C07299=1225.069,224.559,-58.740,-177.166,6.220,148.282
C07300=1225.074,224.310,-58.716,-177.168,6.218,148.282
C07301=1225.078,224.061,-58.690,-177.171,6.216,148.282
C07302=1225.084,223.813,-58.665,-177.173,6.215,148.283
C07303=1225.088,223.563,-58.640,-177.175,6.213,148.283
C07304=1225.092,223.315,-58.615,-177.178,6.211,148.283
C07305=1225.097,223.066,-58.590,-177.181,6.209,148.284
C07306=1225.102,222.818,-58.565,-177.183,6.207,148.284
C07307=1225.105,222.569,-58.541,-177.186,6.206,148.284
C07308=1225.110,222.321,-58.515,-177.188,6.204,148.285
C07309=1225.115,222.072,-58.490,-177.191,6.202,148.285
C07310=1225.120,221.823,-58.465,-177.194,6.200,148.285
C07311=1225.124,221.575,-58.441,-177.196,6.198,148.286
C07312=1225.128,221.325,-58.416,-177.199,6.196,148.286
C07313=1225.133,221.077,-58.390,-177.201,6.195,148.286
C07314=1225.137,220.828,-58.366,-177.204,6.193,148.287
C07315=1225.142,220.579,-58.341,-177.206,6.192,148.287
C07316=1225.146,220.331,-58.315,-177.209,6.190,148.287
C07317=1225.151,220.082,-58.291,-177.212,6.188,148.288
C07318=1225.156,219.833,-58.267,-177.214,6.186,148.288
C07319=1225.160,219.584,-58.242,-177.217,6.184,148.288
C07320=1225.165,219.336,-58.217,-177.219,6.182,148.289
C07321=1225.169,219.087,-58.192,-177.222,6.180,148.289
C07322=1225.174,218.838,-58.167,-177.225,6.178,148.289
C07323=1225.178,218.590,-58.142,-177.227,6.177,148.290
C07324=1225.183,218.341,-58.117,-177.229,6.176,148.290
C07325=1225.187,218.092,-58.093,-177.232,6.174,148.290
C07326=1225.192,217.843,-58.068,-177.235,6.172,148.291
C07327=1225.197,217.594,-58.044,-177.237,6.170,148.291
C07328=1225.201,217.347,-58.019,-177.240,6.168,148.291
C07329=1225.206,217.097,-57.994,-177.243,6.166,148.292
C07330=1225.210,216.849,-57.970,-177.245,6.164,148.292
C07331=1225.214,216.599,-57.945,-177.248,6.163,148.292
C07332=1225.219,216.351,-57.921,-177.250,6.162,148.293
C07333=1225.224,216.102,-57.896,-177.252,6.160,148.293
C07334=1225.228,215.853,-57.870,-177.255,6.158,148.293
C07335=1225.233,215.605,-57.846,-177.258,6.156,148.294
C07336=1225.238,215.356,-57.821,-177.260,6.154,148.294
C07337=1225.242,215.107,-57.797,-177.263,6.152,148.294
C07338=1225.247,214.858,-57.772,-177.266,6.150,148.295
C07339=1225.251,214.610,-57.748,-177.268,6.149,148.295
C07340=1225.256,214.361,-57.723,-177.271,6.147,148.295
C07341=1225.260,214.112,-57.699,-177.273,6.146,148.296
C07342=1225.265,213.863,-57.674,-177.276,6.144,148.296
C07343=1225.269,213.614,-57.650,-177.278,6.142,148.296
C07344=1225.274,213.366,-57.625,-177.281,6.140,148.297
C07345=1225.278,213.117,-57.601,-177.283,6.138,148.297
C07346=1225.283,212.869,-57.577,-177.286,6.136,148.297
C07347=1225.287,212.619,-57.552,-177.289,6.135,148.298
C07348=1225.292,212.371,-57.528,-177.291,6.134,148.298
C07349=1225.297,212.122,-57.503,-177.293,6.132,148.298
C07350=1225.301,211.851,-57.476,-177.296,6.130,148.299
C07351=1225.306,211.581,-57.450,-177.299,6.127,148.299
C07352=1225.311,211.311,-57.423,-177.302,6.125,148.299
C07353=1225.316,211.040,-57.397,-177.305,6.124,148.300
C07354=1225.321,210.792,-57.373,-177.308,6.122,148.300
C07355=1225.325,210.543,-57.348,-177.310,6.121,148.301
C07356=1225.330,210.294,-57.324,-177.312,6.119,148.301
C07357=1225.335,210.046,-57.300,-177.315,6.117,148.301
C07358=1225.339,209.797,-57.276,-177.318,6.115,148.302
C07359=1225.343,209.548,-57.251,-177.320,6.113,148.302
C07360=1225.349,209.299,-57.227,-177.323,6.112,148.302
C07361=1225.353,209.050,-57.203,-177.325,6.111,148.303
C07362=1225.357,208.802,-57.179,-177.328,6.109,148.303
C07363=1225.362,208.552,-57.154,-177.330,6.107,148.303
C07364=1225.366,208.304,-57.130,-177.333,6.105,148.304
C07365=1225.371,208.056,-57.106,-177.336,6.103,148.304
C07366=1225.376,207.806,-57.082,-177.338,6.101,148.304
C07367=1225.380,207.558,-57.058,-177.340,6.100,148.305
C07368=1225.384,207.309,-57.033,-177.343,6.098,148.305
C07369=1225.389,207.060,-57.009,-177.346,6.097,148.305
C07370=1225.394,206.811,-56.985,-177.349,6.095,148.306
C07371=1225.398,206.563,-56.961,-177.351,6.093,148.306
C07372=1225.403,206.314,-56.937,-177.354,6.091,148.307
C07373=1225.408,206.065,-56.912,-177.356,6.090,148.307
C07374=1225.412,205.816,-56.889,-177.359,6.088,148.307
C07375=1225.416,205.567,-56.865,-177.361,6.087,148.308
C07376=1225.421,205.319,-56.841,-177.364,6.085,148.308
C07377=1225.426,205.069,-56.817,-177.367,6.083,148.308
C07378=1225.431,204.821,-56.793,-177.369,6.081,148.309
C07379=1225.435,204.573,-56.768,-177.371,6.080,148.309
C07380=1225.439,204.323,-56.745,-177.374,6.078,148.309
C07381=1225.444,204.075,-56.721,-177.377,6.076,148.310
C07382=1225.449,203.825,-56.697,-177.379,6.074,148.310
C07383=1225.453,203.577,-56.673,-177.382,6.073,148.311
C07384=1225.458,203.328,-56.649,-177.384,6.072,148.311
C07385=1225.463,203.079,-56.625,-177.387,6.070,148.311
C07386=1225.467,202.831,-56.601,-177.390,6.068,148.312
C07387=1225.471,202.581,-56.577,-177.392,6.066,148.312
C07388=1225.476,202.332,-56.553,-177.395,6.065,148.312
C07389=1225.481,202.083,-56.529,-177.397,6.063,148.313
C07390=1225.485,201.835,-56.505,-177.400,6.062,148.313
C07391=1225.490,201.587,-56.481,-177.402,6.060,148.313
C07392=1225.494,201.338,-56.458,-177.405,6.058,148.314
C07393=1225.499,201.089,-56.434,-177.407,6.057,148.314
C07394=1225.503,200.840,-56.410,-177.410,6.055,148.315
C07395=1225.508,200.592,-56.386,-177.413,6.054,148.315
C07396=1225.513,200.343,-56.363,-177.415,6.052,148.315
C07397=1225.518,200.093,-56.339,-177.418,6.050,148.316
C07398=1225.522,199.844,-56.315,-177.420,6.049,148.316
C07399=1225.526,199.595,-56.291,-177.423,6.047,148.316
C07400=1225.531,199.347,-56.267,-177.425,6.045,148.317
C07401=1225.536,199.098,-56.244,-177.428,6.043,148.317
C07402=1225.540,198.849,-56.220,-177.430,6.042,148.317
C07403=1225.545,198.600,-56.196,-177.433,6.040,148.318
C07404=1225.549,198.351,-56.173,-177.436,6.039,148.318
C07405=1225.554,198.103,-56.149,-177.439,6.037,148.319
C07406=1225.558,197.854,-56.126,-177.441,6.035,148.319
C07407=1225.563,197.605,-56.102,-177.443,6.034,148.319
C07408=1225.568,197.356,-56.078,-177.446,6.032,148.320
C07409=1225.572,197.107,-56.055,-177.449,6.030,148.320
C07410=1225.577,196.858,-56.031,-177.451,6.029,148.320
C07411=1225.581,196.610,-56.007,-177.453,6.028,148.321
C07412=1225.586,196.361,-55.984,-177.456,6.026,148.321
C07413=1225.591,196.112,-55.961,-177.459,6.024,148.322
C07414=1225.595,195.863,-55.937,-177.462,6.022,148.322
C07415=1225.600,195.614,-55.913,-177.464,6.021,148.322
C07416=1225.605,195.365,-55.890,-177.466,6.020,148.323
C07417=1225.609,195.116,-55.867,-177.469,6.018,148.323
C07418=1225.614,194.868,-55.842,-177.472,6.016,148.323
C07419=1225.618,194.619,-55.819,-177.474,6.015,148.324
C07420=1225.623,194.370,-55.796,-177.477,6.013,148.324
C07421=1225.628,194.121,-55.772,-177.480,6.011,148.325
C07422=1225.632,193.872,-55.749,-177.482,6.010,148.325
C07423=1225.636,193.624,-55.726,-177.484,6.009,148.325
C07424=1225.641,193.375,-55.702,-177.487,6.007,148.326
C07425=1225.645,193.126,-55.679,-177.490,6.005,148.326
C07426=1225.650,192.877,-55.655,-177.492,6.004,148.327
C07427=1225.655,192.628,-55.632,-177.495,6.002,148.327
C07428=1225.660,192.379,-55.609,-177.497,6.001,148.327
C07429=1225.665,192.131,-55.585,-177.500,5.999,148.328
C07430=1225.669,191.882,-55.562,-177.502,5.998,148.328
C07431=1225.673,191.633,-55.539,-177.505,5.996,148.328
C07432=1225.678,191.384,-55.516,-177.507,5.994,148.329
C07433=1225.683,191.135,-55.492,-177.511,5.993,148.329
C07434=1225.687,190.886,-55.469,-177.513,5.992,148.330
C07435=1225.692,190.637,-55.445,-177.515,5.990,148.330
C07436=1225.697,190.388,-55.422,-177.518,5.988,148.330
C07437=1225.701,190.139,-55.399,-177.520,5.987,148.331
C07438=1225.705,189.890,-55.376,-177.523,5.985,148.331
C07439=1225.711,189.642,-55.353,-177.526,5.983,148.332
C07440=1225.715,189.393,-55.330,-177.528,5.982,148.332
C07441=1225.720,189.144,-55.306,-177.530,5.981,148.333
C07442=1225.724,188.895,-55.284,-177.533,5.979,148.333
C07443=1225.729,188.646,-55.260,-177.536,5.977,148.333
C07444=1225.733,188.397,-55.237,-177.538,5.976,148.334
C07445=1225.738,188.148,-55.213,-177.541,5.974,148.334
C07446=1225.742,187.899,-55.191,-177.544,5.973,148.334
C07447=1225.747,187.651,-55.168,-177.546,5.972,148.335
C07448=1225.752,187.402,-55.144,-177.548,5.970,148.335
C07449=1225.757,187.153,-55.121,-177.551,5.968,148.336
C07450=1225.761,186.904,-55.098,-177.554,5.966,148.336
C07451=1225.765,186.655,-55.075,-177.556,5.965,148.337
C07452=1225.770,186.406,-55.051,-177.559,5.964,148.337
C07453=1225.775,186.157,-55.030,-177.562,5.962,148.337
C07454=1225.779,185.888,-55.004,-177.564,5.960,148.338
C07455=1225.785,185.618,-54.979,-177.567,5.959,148.338
C07456=1225.789,185.348,-54.954,-177.569,5.957,148.339
C07457=1225.795,185.079,-54.929,-177.573,5.956,148.339
C07458=1225.799,184.830,-54.906,-177.575,5.954,148.339
C07459=1225.804,184.581,-54.884,-177.578,5.952,148.340
C07460=1225.809,184.332,-54.861,-177.580,5.951,148.340
C07461=1225.814,184.083,-54.837,-177.583,5.949,148.341
C07462=1225.818,183.834,-54.815,-177.586,5.948,148.341
C07463=1225.823,183.586,-54.792,-177.588,5.947,148.342
C07464=1225.828,183.336,-54.769,-177.590,5.945,148.342
C07465=1225.832,183.087,-54.746,-177.593,5.943,148.342
C07466=1225.837,182.838,-54.723,-177.595,5.942,148.343
C07467=1225.841,182.590,-54.700,-177.598,5.941,148.343
C07468=1225.846,182.341,-54.678,-177.601,5.939,148.344
C07469=1225.851,182.092,-54.654,-177.603,5.938,148.344
C07470=1225.855,181.843,-54.632,-177.606,5.936,148.344
C07471=1225.860,181.593,-54.609,-177.609,5.934,148.345
C07472=1225.864,181.345,-54.587,-177.611,5.933,148.345
C07473=1225.869,181.096,-54.563,-177.614,5.932,148.346
C07474=1225.873,180.847,-54.541,-177.616,5.930,148.346
C07475=1225.878,180.598,-54.518,-177.618,5.929,148.346
C07476=1225.883,180.350,-54.496,-177.621,5.927,148.347
C07477=1225.888,180.100,-54.473,-177.624,5.925,148.347
C07478=1225.892,179.851,-54.450,-177.626,5.924,148.348
C07479=1225.897,179.603,-54.427,-177.629,5.923,148.348
C07480=1225.901,179.354,-54.405,-177.631,5.922,148.349
C07481=1225.906,179.105,-54.382,-177.634,5.920,148.349
C07482=1225.910,178.855,-54.360,-177.637,5.918,148.349
C07483=1225.915,178.607,-54.337,-177.639,5.917,148.350
C07484=1225.920,178.358,-54.315,-177.642,5.916,148.350
C07485=1225.924,178.109,-54.291,-177.645,5.914,148.351
C07486=1225.929,177.861,-54.269,-177.647,5.913,148.351
C07487=1225.934,177.611,-54.246,-177.649,5.911,148.351
C07488=1225.938,177.362,-54.223,-177.652,5.909,148.352
C07489=1225.944,177.113,-54.201,-177.655,5.908,148.352
C07490=1225.947,176.865,-54.178,-177.657,5.907,148.353
C07491=1225.952,176.615,-54.156,-177.659,5.906,148.353
C07492=1225.957,176.367,-54.133,-177.662,5.904,148.353
C07493=1225.961,176.118,-54.111,-177.665,5.902,148.354
C07494=1225.966,175.868,-54.089,-177.667,5.901,148.354
C07495=1225.971,175.620,-54.066,-177.670,5.899,148.355
C07496=1225.976,175.370,-54.044,-177.673,5.898,148.355
C07497=1225.980,175.122,-54.021,-177.675,5.897,148.356
C07498=1225.985,174.873,-53.999,-177.678,5.895,148.356
C07499=1225.989,174.624,-53.976,-177.680,5.894,148.356
C07500=1225.994,174.375,-53.954,-177.683,5.893,148.357
C07501=1225.999,174.126,-53.932,-177.686,5.891,148.357
C07502=1226.003,173.877,-53.909,-177.688,5.890,148.358
C07503=1226.008,173.628,-53.887,-177.690,5.888,148.358
C07504=1226.013,173.379,-53.864,-177.693,5.887,148.359
C07505=1226.017,173.130,-53.842,-177.696,5.885,148.359
C07506=1226.022,172.881,-53.820,-177.698,5.884,148.359
C07507=1226.027,172.632,-53.797,-177.700,5.883,148.360
C07508=1226.032,172.384,-53.775,-177.704,5.881,148.360
C07509=1226.036,172.134,-53.753,-177.706,5.880,148.361
C07510=1226.041,171.885,-53.730,-177.708,5.878,148.361
C07511=1226.045,171.637,-53.708,-177.711,5.877,148.362
C07512=1226.050,171.387,-53.686,-177.713,5.876,148.362
C07513=1226.055,171.138,-53.664,-177.716,5.874,148.363
C07514=1226.060,170.889,-53.641,-177.718,5.873,148.363
C07515=1226.064,170.641,-53.619,-177.721,5.871,148.363
C07516=1226.068,170.392,-53.597,-177.724,5.870,148.364
C07517=1226.073,170.142,-53.574,-177.726,5.869,148.364
C07518=1226.078,169.893,-53.553,-177.729,5.867,148.365
C07519=1226.082,169.645,-53.530,-177.731,5.866,148.365
C07520=1226.087,169.396,-53.508,-177.734,5.864,148.366
C07521=1226.092,169.146,-53.486,-177.737,5.862,148.366
C07522=1226.097,168.898,-53.464,-177.739,5.862,148.367
C07523=1226.101,168.648,-53.442,-177.742,5.860,148.367
C07524=1226.106,168.400,-53.420,-177.744,5.859,148.367
C07525=1226.110,168.151,-53.397,-177.747,5.858,148.368
C07526=1226.116,167.902,-53.375,-177.749,5.857,148.368
C07527=1226.120,167.653,-53.353,-177.752,5.855,148.369
C07528=1226.125,167.404,-53.331,-177.755,5.853,148.369
C07529=1226.129,167.155,-53.309,-177.757,5.852,148.370
C07530=1226.134,166.906,-53.288,-177.760,5.850,148.370
C07531=1226.139,166.656,-53.265,-177.762,5.849,148.370
C07532=1226.144,166.408,-53.243,-177.765,5.848,148.371
C07533=1226.148,166.158,-53.221,-177.767,5.847,148.371
C07534=1226.153,165.910,-53.200,-177.770,5.845,148.372
C07535=1226.157,165.660,-53.178,-177.772,5.844,148.372
C07536=1226.162,165.412,-53.155,-177.775,5.843,148.373
C07537=1226.166,165.163,-53.133,-177.778,5.841,148.373
C07538=1226.171,164.914,-53.111,-177.780,5.840,148.374
C07539=1226.176,164.665,-53.089,-177.783,5.838,148.374
C07540=1226.181,164.416,-53.067,-177.785,5.837,148.374
C07541=1226.185,164.167,-53.045,-177.788,5.836,148.375
C07542=1226.190,163.918,-53.023,-177.790,5.835,148.375
C07543=1226.195,163.669,-53.002,-177.793,5.833,148.376
C07544=1226.199,163.419,-52.980,-177.796,5.832,148.376
C07545=1226.204,163.171,-52.959,-177.798,5.830,148.377
C07546=1226.208,162.922,-52.937,-177.801,5.829,148.377
C07547=1226.213,162.673,-52.915,-177.803,5.828,148.378
C07548=1226.218,162.424,-52.893,-177.806,5.826,148.378
C07549=1226.222,162.175,-52.871,-177.808,5.825,148.378
C07550=1226.227,161.926,-52.850,-177.811,5.824,148.379
C07551=1226.232,161.677,-52.828,-177.813,5.823,148.379
C07552=1226.236,161.428,-52.806,-177.816,5.821,148.380
C07553=1226.241,161.179,-52.784,-177.819,5.820,148.380
C07554=1226.246,160.930,-52.763,-177.821,5.818,148.381
C07555=1226.251,160.681,-52.741,-177.823,5.817,148.381
C07556=1226.255,160.432,-52.719,-177.827,5.816,148.382
C07557=1226.260,160.183,-52.697,-177.829,5.815,148.382
C07558=1226.265,159.914,-52.674,-177.831,5.813,148.383
C07559=1226.271,159.645,-52.650,-177.835,5.812,148.383
C07560=1226.275,159.376,-52.627,-177.838,5.810,148.384
C07561=1226.281,159.107,-52.604,-177.840,5.809,148.384
C07562=1226.285,158.857,-52.582,-177.842,5.807,148.384
C07563=1226.290,158.609,-52.560,-177.845,5.807,148.385
C07564=1226.294,158.359,-52.538,-177.848,5.805,148.385
C07565=1226.299,158.110,-52.517,-177.850,5.804,148.386
C07566=1226.304,157.861,-52.495,-177.853,5.802,148.386
C07567=1226.308,157.612,-52.474,-177.855,5.801,148.387
C07568=1226.313,157.364,-52.452,-177.858,5.800,148.387
C07569=1226.318,157.114,-52.431,-177.860,5.799,148.388
C07570=1226.322,156.865,-52.409,-177.863,5.797,148.388
C07571=1226.327,156.616,-52.388,-177.866,5.796,148.389
C07572=1226.332,156.367,-52.367,-177.868,5.795,148.389
C07573=1226.336,156.118,-52.345,-177.870,5.794,148.390
C07574=1226.341,155.869,-52.323,-177.873,5.792,148.390
C07575=1226.346,155.620,-52.302,-177.876,5.791,148.391
C07576=1226.351,155.372,-52.281,-177.879,5.790,148.391
C07577=1226.355,155.122,-52.259,-177.881,5.789,148.392
C07578=1226.360,154.873,-52.238,-177.883,5.787,148.392
C07579=1226.365,154.624,-52.216,-177.886,5.786,148.393
C07580=1226.370,154.374,-52.195,-177.889,5.784,148.393
C07581=1226.374,154.126,-52.173,-177.891,5.784,148.394
C07582=1226.378,153.877,-52.152,-177.894,5.782,148.394
C07583=1226.384,153.628,-52.131,-177.896,5.781,148.394
C07584=1226.388,153.379,-52.109,-177.899,5.779,148.395
C07585=1226.393,153.130,-52.088,-177.901,5.778,148.395
C07586=1226.398,152.881,-52.066,-177.904,5.777,148.396
C07587=1226.403,152.632,-52.045,-177.907,5.776,148.396
C07588=1226.407,152.383,-52.024,-177.909,5.774,148.397
C07589=1226.412,152.133,-52.003,-177.912,5.773,148.397
C07590=1226.417,151.885,-51.981,-177.915,5.772,148.398
C07591=1226.422,151.635,-51.960,-177.917,5.771,148.398
C07592=1226.425,151.386,-51.939,-177.919,5.770,148.399
C07593=1226.431,151.137,-51.918,-177.922,5.768,148.399
C07594=1226.435,150.889,-51.896,-177.924,5.767,148.400
C07595=1226.441,150.639,-51.875,-177.927,5.766,148.400
C07596=1226.444,150.390,-51.854,-177.929,5.765,148.400
C07597=1226.449,150.141,-51.833,-177.932,5.763,148.401
C07598=1226.454,149.892,-51.811,-177.935,5.762,148.401
C07599=1226.459,149.643,-51.791,-177.938,5.761,148.402
C07600=1226.464,149.394,-51.770,-177.940,5.760,148.402
C07601=1226.468,149.145,-51.748,-177.942,5.758,148.403
C07602=1226.473,148.896,-51.727,-177.945,5.757,148.403
C07603=1226.478,148.647,-51.706,-177.948,5.755,148.404
C07604=1226.483,148.398,-51.685,-177.950,5.755,148.404
C07605=1226.488,148.149,-51.664,-177.952,5.754,148.405
C07606=1226.491,147.900,-51.642,-177.956,5.752,148.405
C07607=1226.496,147.650,-51.621,-177.958,5.751,148.406
C07608=1226.502,147.401,-51.600,-177.960,5.750,148.406
C07609=1226.506,147.153,-51.579,-177.963,5.749,148.407
C07610=1226.511,146.904,-51.558,-177.966,5.747,148.407
C07611=1226.515,146.655,-51.538,-177.968,5.746,148.408
C07612=1226.520,146.405,-51.517,-177.971,5.745,148.408
C07613=1226.525,146.156,-51.495,-177.973,5.744,148.409
C07614=1226.529,145.907,-51.475,-177.976,5.743,148.409
C07615=1226.534,145.658,-51.454,-177.978,5.741,148.410
C07616=1226.539,145.409,-51.433,-177.981,5.741,148.410
C07617=1226.544,145.160,-51.412,-177.983,5.739,148.411
C07618=1226.549,144.911,-51.391,-177.986,5.738,148.411
C07619=1226.553,144.661,-51.370,-177.989,5.736,148.412
C07620=1226.558,144.412,-51.349,-177.991,5.736,148.412
C07621=1226.562,144.164,-51.328,-177.993,5.735,148.413
C07622=1226.567,143.914,-51.307,-177.996,5.733,148.413
C07623=1226.572,143.665,-51.286,-177.999,5.732,148.414
C07624=1226.577,143.416,-51.266,-178.001,5.730,148.414
C07625=1226.582,143.167,-51.245,-178.004,5.730,148.415
C07626=1226.586,142.918,-51.224,-178.007,5.728,148.415
C07627=1226.591,142.669,-51.202,-178.009,5.727,148.416
C07628=1226.595,142.420,-51.182,-178.011,5.726,148.416
C07629=1226.600,142.170,-51.161,-178.015,5.725,148.417
C07630=1226.605,141.922,-51.140,-178.017,5.724,148.417
C07631=1226.610,141.672,-51.119,-178.020,5.722,148.418
C07632=1226.614,141.423,-51.099,-178.022,5.721,148.418
C07633=1226.620,141.174,-51.078,-178.024,5.720,148.419
C07634=1226.624,140.925,-51.058,-178.027,5.719,148.419
C07635=1226.629,140.676,-51.037,-178.029,5.718,148.420
C07636=1226.633,140.428,-51.016,-178.032,5.716,148.420
C07637=1226.638,140.179,-50.995,-178.035,5.715,148.421
C07638=1226.643,139.929,-50.974,-178.037,5.715,148.421
C07639=1226.647,139.680,-50.954,-178.040,5.713,148.422
C07640=1226.653,139.431,-50.933,-178.042,5.712,148.422
C07641=1226.657,139.182,-50.913,-178.045,5.711,148.423
C07642=1226.662,138.933,-50.892,-178.048,5.710,148.423
C07643=1226.667,138.684,-50.871,-178.050,5.709,148.424
C07644=1226.671,138.435,-50.851,-178.053,5.707,148.424
C07645=1226.676,138.186,-50.830,-178.055,5.707,148.425
C07646=1226.681,137.937,-50.810,-178.058,5.705,148.425
C07647=1226.686,137.688,-50.789,-178.060,5.704,148.426
C07648=1226.691,137.438,-50.769,-178.062,5.703,148.426
C07649=1226.695,137.189,-50.749,-178.066,5.702,148.427
C07650=1226.700,136.940,-50.728,-178.068,5.701,148.427
C07651=1226.705,136.691,-50.707,-178.070,5.700,148.428
C07652=1226.710,136.442,-50.686,-178.073,5.698,148.428
C07653=1226.714,136.193,-50.666,-178.076,5.698,148.429
C07654=1226.719,135.944,-50.646,-178.078,5.696,148.429
C07655=1226.724,135.694,-50.625,-178.081,5.695,148.430
C07656=1226.728,135.445,-50.604,-178.083,5.694,148.430
C07657=1226.733,135.196,-50.584,-178.086,5.693,148.431
C07658=1226.738,134.947,-50.564,-178.088,5.692,148.431
C07659=1226.743,134.698,-50.543,-178.091,5.691,148.432
C07660=1226.747,134.449,-50.523,-178.094,5.689,148.432
C07661=1226.752,134.199,-50.502,-178.096,5.689,148.433
C07662=1226.757,133.931,-50.481,-178.099,5.687,148.433
C07663=1226.762,133.662,-50.458,-178.101,5.686,148.434
C07664=1226.767,133.393,-50.436,-178.105,5.685,148.434
C07665=1226.772,133.125,-50.415,-178.107,5.684,148.435
C07666=1226.777,132.875,-50.394,-178.110,5.682,148.435
C07667=1226.782,132.627,-50.373,-178.112,5.682,148.436
C07668=1226.787,132.377,-50.354,-178.115,5.681,148.436
C07669=1226.791,132.128,-50.333,-178.118,5.679,148.437
C07670=1226.796,131.879,-50.312,-178.120,5.678,148.437
C07671=1226.801,131.630,-50.292,-178.123,5.677,148.438
C07672=1226.806,131.381,-50.273,-178.125,5.676,148.438
C07673=1226.810,131.132,-50.252,-178.128,5.675,148.439
C07674=1226.816,130.883,-50.231,-178.130,5.673,148.439
C07675=1226.820,130.633,-50.212,-178.133,5.673,148.440
C07676=1226.825,130.384,-50.191,-178.135,5.672,148.440
C07677=1226.829,130.135,-50.171,-178.138,5.670,148.441
C07678=1226.834,129.886,-50.151,-178.140,5.669,148.442
C07679=1226.839,129.636,-50.130,-178.143,5.669,148.442
C07680=1226.843,129.387,-50.110,-178.146,5.667,148.443
C07681=1226.849,129.139,-50.091,-178.148,5.666,148.443
C07682=1226.853,128.890,-50.070,-178.150,5.665,148.444
C07683=1226.858,128.640,-50.050,-178.154,5.664,148.444
C07684=1226.862,128.391,-50.030,-178.156,5.663,148.445
C07685=1226.867,128.142,-50.010,-178.158,5.662,148.445
C07686=1226.872,127.892,-49.989,-178.161,5.661,148.446
C07687=1226.877,127.643,-49.969,-178.164,5.660,148.446
C07688=1226.882,127.395,-49.950,-178.166,5.659,148.447
C07689=1226.887,127.146,-49.929,-178.169,5.657,148.447
C07690=1226.891,126.897,-49.909,-178.171,5.657,148.448
C07691=1226.896,126.647,-49.889,-178.174,5.656,148.448
C07692=1226.900,126.398,-49.869,-178.177,5.654,148.449
C07693=1226.905,126.149,-49.849,-178.179,5.653,148.449
C07694=1226.910,125.900,-49.829,-178.181,5.653,148.450
C07695=1226.915,125.650,-49.809,-178.184,5.652,148.450
C07696=1226.920,125.401,-49.789,-178.187,5.650,148.451
C07697=1226.925,125.152,-49.769,-178.189,5.649,148.451
C07698=1226.929,124.903,-49.749,-178.191,5.649,148.452
C07699=1226.934,124.654,-49.729,-178.195,5.647,148.453
C07700=1226.939,124.405,-49.710,-178.197,5.646,148.453
C07701=1226.944,124.156,-49.689,-178.199,5.646,148.454
C07702=1226.948,123.906,-49.670,-178.202,5.644,148.454
C07703=1226.953,123.657,-49.649,-178.205,5.643,148.455
C07704=1226.958,123.408,-49.630,-178.207,5.642,148.455
C07705=1226.963,123.159,-49.610,-178.210,5.641,148.456
C07706=1226.967,122.910,-49.590,-178.212,5.640,148.456
C07707=1226.972,122.660,-49.570,-178.215,5.639,148.457
C07708=1226.977,122.412,-49.550,-178.217,5.638,148.457
C07709=1226.982,122.162,-49.531,-178.220,5.637,148.458
C07710=1226.987,121.913,-49.511,-178.223,5.636,148.458
C07711=1226.991,121.664,-49.491,-178.225,5.635,148.459
C07712=1226.996,121.415,-49.471,-178.228,5.634,148.459
C07713=1227.001,121.165,-49.452,-178.230,5.633,148.460
C07714=1227.006,120.916,-49.431,-178.233,5.632,148.461
C07715=1227.010,120.667,-49.412,-178.236,5.631,148.461
C07716=1227.016,120.418,-49.392,-178.238,5.630,148.462
C07717=1227.020,120.169,-49.372,-178.240,5.629,148.462
C07718=1227.025,119.919,-49.352,-178.243,5.628,148.463
C07719=1227.030,119.671,-49.333,-178.246,5.626,148.463
C07720=1227.035,119.422,-49.313,-178.248,5.626,148.464
C07721=1227.039,119.172,-49.294,-178.250,5.625,148.464
C07722=1227.043,118.923,-49.274,-178.253,5.624,148.465
C07723=1227.049,118.674,-49.255,-178.256,5.622,148.465
C07724=1227.053,118.425,-49.234,-178.258,5.622,148.466
C07725=1227.058,118.175,-49.215,-178.260,5.621,148.466
C07726=1227.063,117.927,-49.195,-178.264,5.619,148.467
C07727=1227.068,117.677,-49.176,-178.266,5.618,148.467
C07728=1227.073,117.427,-49.156,-178.268,5.618,148.468
C07729=1227.078,117.179,-49.136,-178.271,5.617,148.469
C07730=1227.082,116.930,-49.117,-178.274,5.615,148.469
C07731=1227.086,116.680,-49.097,-178.276,5.615,148.470
C07732=1227.092,116.431,-49.078,-178.278,5.614,148.470
C07733=1227.097,116.182,-49.058,-178.281,5.613,148.471
C07734=1227.101,115.932,-49.039,-178.284,5.612,148.471
C07735=1227.107,115.683,-49.020,-178.286,5.611,148.472
C07736=1227.110,115.435,-49.000,-178.289,5.610,148.472
C07737=1227.115,115.185,-48.980,-178.291,5.609,148.473
C07738=1227.120,114.936,-48.961,-178.294,5.608,148.473
C07739=1227.125,114.687,-48.941,-178.297,5.607,148.474
C07740=1227.130,114.437,-48.921,-178.299,5.606,148.475
C07741=1227.135,114.189,-48.903,-178.302,5.606,148.475
C07742=1227.139,113.939,-48.883,-178.304,5.604,148.476
C07743=1227.145,113.690,-48.864,-178.307,5.603,148.476
C07744=1227.149,113.441,-48.844,-178.309,5.603,148.477
C07745=1227.154,113.191,-48.825,-178.312,5.602,148.477
C07746=1227.159,112.943,-48.806,-178.315,5.600,148.478
C07747=1227.163,112.693,-48.786,-178.317,5.599,148.478
C07748=1227.169,112.444,-48.767,-178.319,5.599,148.479
C07749=1227.174,112.195,-48.747,-178.322,5.598,148.480
C07750=1227.178,111.945,-48.728,-178.325,5.596,148.480
C07751=1227.183,111.696,-48.709,-178.327,5.595,148.481
C07752=1227.188,111.447,-48.689,-178.330,5.595,148.481
C07753=1227.193,111.198,-48.670,-178.332,5.594,148.482
C07754=1227.197,110.949,-48.651,-178.335,5.592,148.482
C07755=1227.202,110.699,-48.631,-178.337,5.591,148.483
C07756=1227.207,110.450,-48.612,-178.340,5.591,148.483
C07757=1227.211,110.201,-48.593,-178.343,5.590,148.484
C07758=1227.216,109.952,-48.574,-178.345,5.588,148.484
C07759=1227.221,109.703,-48.554,-178.348,5.588,148.485
C07760=1227.226,109.454,-48.535,-178.351,5.587,148.486
C07761=1227.231,109.204,-48.516,-178.353,5.586,148.486
C07762=1227.236,108.955,-48.497,-178.355,5.586,148.487
C07763=1227.240,108.706,-48.478,-178.358,5.584,148.487
C07764=1227.246,108.457,-48.459,-178.361,5.583,148.488
C07765=1227.250,108.207,-48.439,-178.363,5.583,148.488
C07766=1227.254,107.939,-48.418,-178.366,5.582,148.489
C07767=1227.260,107.670,-48.398,-178.369,5.580,148.489
C07768=1227.265,107.402,-48.377,-178.371,5.580,148.490
C07769=1227.271,107.134,-48.357,-178.374,5.578,148.491
C07770=1227.275,106.884,-48.337,-178.377,5.578,148.491
C07771=1227.280,106.635,-48.319,-178.379,5.577,148.492
C07772=1227.285,106.385,-48.299,-178.382,5.576,148.492
C07773=1227.290,106.137,-48.281,-178.384,5.575,148.493
C07774=1227.294,105.887,-48.261,-178.387,5.574,148.493
C07775=1227.300,105.639,-48.242,-178.390,5.573,148.494
C07776=1227.304,105.389,-48.223,-178.392,5.572,148.495
C07777=1227.309,105.140,-48.204,-178.394,5.571,148.495
C07778=1227.313,104.890,-48.185,-178.397,5.571,148.496
C07779=1227.319,104.641,-48.166,-178.400,5.569,148.496
C07780=1227.323,104.392,-48.147,-178.402,5.568,148.497
C07781=1227.328,104.143,-48.128,-178.405,5.568,148.498
C07782=1227.333,103.894,-48.109,-178.407,5.567,148.498
C07783=1227.338,103.644,-48.090,-178.410,5.566,148.499
C07784=1227.343,103.396,-48.072,-178.413,5.565,148.499
C07785=1227.347,103.146,-48.052,-178.415,5.564,148.500
C07786=1227.352,102.897,-48.034,-178.417,5.563,148.500
C07787=1227.357,102.647,-48.014,-178.420,5.563,148.501
C07788=1227.362,102.399,-47.996,-178.423,5.562,148.502
C07789=1227.367,102.149,-47.977,-178.425,5.560,148.502
C07790=1227.371,101.900,-47.958,-178.428,5.560,148.503
C07791=1227.377,101.650,-47.940,-178.431,5.559,148.503
C07792=1227.381,101.401,-47.921,-178.433,5.558,148.504
C07793=1227.386,101.152,-47.901,-178.435,5.557,148.504
C07794=1227.391,100.902,-47.883,-178.438,5.557,148.505
C07795=1227.396,100.654,-47.864,-178.441,5.555,148.505
C07796=1227.400,100.404,-47.845,-178.443,5.554,148.506
C07797=1227.406,100.155,-47.826,-178.446,5.554,148.507
C07798=1227.410,99.906,-47.807,-178.448,5.553,148.507
C07799=1227.415,99.656,-47.789,-178.451,5.552,148.508
C07800=1227.420,99.408,-47.770,-178.454,5.551,148.508
C07801=1227.424,99.158,-47.751,-178.456,5.550,148.509
C07802=1227.430,98.909,-47.732,-178.459,5.549,148.509
C07803=1227.434,98.660,-47.714,-178.461,5.549,148.510
C07804=1227.439,98.410,-47.694,-178.463,5.548,148.511
C07805=1227.444,98.161,-47.676,-178.466,5.547,148.511
C07806=1227.449,97.912,-47.658,-178.469,5.546,148.512
C07807=1227.454,97.662,-47.639,-178.471,5.545,148.512
C07808=1227.458,97.414,-47.620,-178.474,5.544,148.513
C07809=1227.463,97.164,-47.602,-178.477,5.543,148.514
C07810=1227.468,96.914,-47.583,-178.479,5.542,148.514
C07811=1227.473,96.666,-47.564,-178.481,5.542,148.515
C07812=1227.478,96.417,-47.546,-178.484,5.541,148.515
C07813=1227.483,96.167,-47.527,-178.487,5.539,148.516
C07814=1227.488,95.918,-47.509,-178.489,5.539,148.516
C07815=1227.492,95.669,-47.490,-178.492,5.538,148.517
C07816=1227.497,95.419,-47.471,-178.494,5.538,148.518
C07817=1227.502,95.170,-47.453,-178.497,5.537,148.518
C07818=1227.507,94.921,-47.435,-178.499,5.536,148.519
C07819=1227.512,94.671,-47.416,-178.502,5.535,148.519
C07820=1227.517,94.422,-47.398,-178.504,5.534,148.520
C07821=1227.521,94.173,-47.379,-178.507,5.533,148.520
C07822=1227.526,93.923,-47.360,-178.510,5.532,148.521
C07823=1227.531,93.674,-47.342,-178.512,5.532,148.521
C07824=1227.536,93.425,-47.323,-178.514,5.531,148.522
C07825=1227.540,93.176,-47.305,-178.517,5.530,148.523
C07826=1227.546,92.926,-47.286,-178.520,5.530,148.523
C07827=1227.550,92.678,-47.268,-178.522,5.528,148.524
C07828=1227.555,92.428,-47.250,-178.525,5.527,148.524
C07829=1227.560,92.178,-47.231,-178.528,5.527,148.525
C07830=1227.565,91.930,-47.212,-178.530,5.526,148.526
C07831=1227.570,91.680,-47.194,-178.532,5.525,148.526
C07832=1227.574,91.431,-47.176,-178.535,5.525,148.527
C07833=1227.579,91.181,-47.158,-178.538,5.524,148.528
C07834=1227.584,90.933,-47.138,-178.540,5.523,148.528
C07835=1227.589,90.683,-47.120,-178.543,5.522,148.529
C07836=1227.594,90.433,-47.102,-178.546,5.521,148.529
C07837=1227.599,90.184,-47.084,-178.548,5.520,148.530
C07838=1227.603,89.935,-47.066,-178.550,5.519,148.530
C07839=1227.609,89.686,-47.047,-178.553,5.519,148.531
C07840=1227.613,89.436,-47.029,-178.556,5.518,148.532
C07841=1227.618,89.187,-47.011,-178.558,5.517,148.532
C07842=1227.623,88.938,-46.993,-178.560,5.517,148.533
C07843=1227.628,88.689,-46.975,-178.564,5.515,148.533
C07844=1227.633,88.440,-46.957,-178.566,5.515,148.534
C07845=1227.637,88.190,-46.938,-178.568,5.514,148.534
C07846=1227.642,87.941,-46.919,-178.571,5.513,148.535
C07847=1227.647,87.692,-46.901,-178.574,5.512,148.536
C07848=1227.652,87.443,-46.883,-178.576,5.512,148.536
C07849=1227.657,87.193,-46.865,-178.578,5.511,148.537
C07850=1227.662,86.944,-46.847,-178.581,5.510,148.537
C07851=1227.666,86.694,-46.829,-178.583,5.510,148.538
C07852=1227.671,86.445,-46.811,-178.586,5.508,148.538
C07853=1227.676,86.196,-46.793,-178.589,5.507,148.539
C07854=1227.681,85.947,-46.775,-178.591,5.507,148.540
C07855=1227.686,85.697,-46.756,-178.594,5.506,148.540
C07856=1227.691,85.447,-46.738,-178.596,5.505,148.541
C07857=1227.696,85.198,-46.720,-178.599,5.505,148.542
C07858=1227.701,84.950,-46.701,-178.601,5.504,148.542
C07859=1227.706,84.701,-46.683,-178.604,5.503,148.543
C07860=1227.710,84.451,-46.665,-178.606,5.502,148.543
C07861=1227.715,84.201,-46.647,-178.609,5.502,148.544
C07862=1227.720,83.952,-46.629,-178.611,5.501,148.545
C07863=1227.725,83.703,-46.612,-178.615,5.500,148.545
C07864=1227.730,83.453,-46.594,-178.617,5.499,148.546
C07865=1227.735,83.204,-46.576,-178.619,5.498,148.546
C07866=1227.740,82.955,-46.558,-178.622,5.498,148.547
C07867=1227.745,82.706,-46.540,-178.625,5.497,148.548
C07868=1227.749,82.456,-46.521,-178.627,5.496,148.548
C07869=1227.754,82.207,-46.503,-178.629,5.496,148.549
C07870=1227.759,81.939,-46.484,-178.632,5.495,148.549
C07871=1227.764,81.670,-46.465,-178.635,5.494,148.550
C07872=1227.769,81.402,-46.445,-178.638,5.493,148.551
C07873=1227.774,81.133,-46.426,-178.640,5.492,148.551
C07874=1227.779,80.884,-46.408,-178.643,5.492,148.552
C07875=1227.784,80.635,-46.390,-178.646,5.491,148.553
C07876=1227.789,80.386,-46.373,-178.648,5.490,148.553
C07877=1227.794,80.136,-46.355,-178.650,5.490,148.554
C07878=1227.799,79.887,-46.337,-178.653,5.489,148.554
C07879=1227.804,79.638,-46.319,-178.656,5.488,148.555
C07880=1227.809,79.388,-46.301,-178.658,5.488,148.555
C07881=1227.814,79.139,-46.283,-178.661,5.486,148.556
C07882=1227.819,78.890,-46.265,-178.664,5.486,148.557
C07883=1227.824,78.641,-46.247,-178.666,5.485,148.557
C07884=1227.829,78.392,-46.229,-178.669,5.484,148.558
C07885=1227.834,78.142,-46.212,-178.671,5.483,148.558
C07886=1227.838,77.892,-46.194,-178.674,5.483,148.559
C07887=1227.842,77.643,-46.176,-178.676,5.482,148.560
C07888=1227.847,77.394,-46.158,-178.679,5.482,148.560
C07889=1227.853,77.144,-46.141,-178.681,5.481,148.561
C07890=1227.857,76.895,-46.123,-178.684,5.480,148.562
C07891=1227.862,76.646,-46.105,-178.686,5.479,148.562
C07892=1227.867,76.397,-46.087,-178.689,5.479,148.563
C07893=1227.873,76.147,-46.070,-178.692,5.478,148.564
C07894=1227.877,75.898,-46.052,-178.694,5.477,148.564
C07895=1227.882,75.649,-46.035,-178.696,5.477,148.565
C07896=1227.887,75.399,-46.017,-178.699,5.476,148.565
C07897=1227.892,75.150,-45.999,-178.702,5.476,148.566
C07898=1227.897,74.901,-45.981,-178.704,5.475,148.566
C07899=1227.902,74.651,-45.964,-178.706,5.474,148.567
C07900=1227.906,74.402,-45.947,-178.710,5.473,148.568
C07901=1227.911,74.153,-45.929,-178.712,5.472,148.568
C07902=1227.916,73.903,-45.911,-178.715,5.471,148.569
C07903=1227.921,73.654,-45.893,-178.717,5.471,148.569
C07904=1227.926,73.405,-45.876,-178.720,5.470,148.570
C07905=1227.930,73.155,-45.859,-178.722,5.469,148.571
C07906=1227.935,72.906,-45.841,-178.725,5.469,148.571
C07907=1227.941,72.656,-45.824,-178.727,5.468,148.572
C07908=1227.946,72.407,-45.806,-178.730,5.467,148.572
C07909=1227.950,72.158,-45.788,-178.732,5.467,148.573
C07910=1227.955,71.908,-45.771,-178.735,5.466,148.574
C07911=1227.960,71.659,-45.753,-178.737,5.465,148.574
C07912=1227.965,71.409,-45.736,-178.740,5.465,148.575
C07913=1227.969,71.160,-45.718,-178.742,5.464,148.576
C07914=1227.975,70.911,-45.701,-178.745,5.463,148.576
C07915=1227.980,70.662,-45.683,-178.748,5.463,148.577
C07916=1227.985,70.412,-45.666,-178.750,5.462,148.578
C07917=1227.989,70.164,-45.649,-178.753,5.462,148.578
C07918=1227.995,69.914,-45.632,-178.755,5.461,148.579
C07919=1227.999,69.665,-45.614,-178.758,5.460,148.579
C07920=1228.004,69.415,-45.597,-178.760,5.460,148.580
C07921=1228.009,69.166,-45.579,-178.763,5.459,148.581
C07922=1228.014,68.916,-45.562,-178.765,5.458,148.581
C07923=1228.018,68.667,-45.544,-178.768,5.458,148.582
C07924=1228.023,68.417,-45.527,-178.770,5.457,148.582
C07925=1228.028,68.168,-45.509,-178.773,5.456,148.583
C07926=1228.033,67.919,-45.492,-178.775,5.456,148.584
C07927=1228.038,67.670,-45.475,-178.778,5.455,148.584
C07928=1228.044,67.421,-45.457,-178.781,5.454,148.585
C07929=1228.048,67.171,-45.441,-178.783,5.454,148.585
C07930=1228.053,66.922,-45.423,-178.785,5.453,148.586
C07931=1228.058,66.672,-45.406,-178.788,5.452,148.587
C07932=1228.062,66.423,-45.388,-178.791,5.452,148.587
C07933=1228.068,66.173,-45.371,-178.793,5.451,148.588
C07934=1228.072,65.924,-45.354,-178.796,5.451,148.589
C07935=1228.077,65.675,-45.336,-178.798,5.450,148.589
C07936=1228.083,65.426,-45.319,-178.801,5.449,148.590
C07937=1228.087,65.176,-45.303,-178.803,5.449,148.591
C07938=1228.092,64.927,-45.285,-178.806,5.448,148.591
C07939=1228.097,64.678,-45.268,-178.809,5.447,148.592
C07940=1228.102,64.428,-45.251,-178.811,5.447,148.593
C07941=1228.106,64.179,-45.233,-178.813,5.446,148.593
C07942=1228.112,63.930,-45.216,-178.816,5.445,148.594
C07943=1228.117,63.680,-45.199,-178.819,5.445,148.594
C07944=1228.122,63.430,-45.183,-178.821,5.444,148.595
C07945=1228.126,63.181,-45.165,-178.824,5.444,148.596
C07946=1228.131,62.932,-45.148,-178.827,5.443,148.596
C07947=1228.136,62.682,-45.131,-178.829,5.442,148.597
C07948=1228.141,62.433,-45.114,-178.831,5.441,148.597
C07949=1228.146,62.184,-45.096,-178.834,5.441,148.598
C07950=1228.151,61.935,-45.080,-178.837,5.440,148.599
C07951=1228.156,61.685,-45.062,-178.839,5.440,148.599
C07952=1228.160,61.435,-45.046,-178.842,5.439,148.600
C07953=1228.166,61.187,-45.028,-178.844,5.438,148.600
C07954=1228.170,60.937,-45.011,-178.847,5.438,148.601
C07955=1228.176,60.688,-44.994,-178.849,5.437,148.602
C07956=1228.180,60.438,-44.978,-178.852,5.436,148.602
C07957=1228.185,60.188,-44.960,-178.855,5.436,148.603
C07958=1228.190,59.939,-44.944,-178.857,5.435,148.604
C07959=1228.195,59.690,-44.926,-178.859,5.434,148.604
C07960=1228.200,59.441,-44.909,-178.862,5.434,148.605
C07961=1228.205,59.191,-44.892,-178.865,5.433,148.606
C07962=1228.210,58.942,-44.876,-178.867,5.433,148.606
C07963=1228.215,58.693,-44.859,-178.870,5.432,148.607
C07964=1228.220,58.443,-44.842,-178.872,5.431,148.608
C07965=1228.224,58.193,-44.825,-178.875,5.431,148.608
C07966=1228.230,57.944,-44.808,-178.877,5.430,148.609
C07967=1228.234,57.696,-44.791,-178.879,5.430,148.609
C07968=1228.239,57.446,-44.774,-178.882,5.430,148.610
C07969=1228.244,57.196,-44.757,-178.885,5.429,148.611
C07970=1228.249,56.947,-44.741,-178.887,5.429,148.611
C07971=1228.254,56.698,-44.723,-178.890,5.428,148.612
C07972=1228.259,56.448,-44.707,-178.893,5.427,148.613
C07973=1228.264,56.198,-44.689,-178.895,5.426,148.613
C07974=1228.269,55.931,-44.672,-178.898,5.426,148.614
C07975=1228.274,55.662,-44.654,-178.900,5.426,148.615
C07976=1228.280,55.393,-44.636,-178.904,5.424,148.615
C07977=1228.285,55.125,-44.618,-178.906,5.424,148.616
C07978=1228.291,54.876,-44.601,-178.909,5.423,148.617
C07979=1228.295,54.626,-44.584,-178.910,5.423,148.617
C07980=1228.300,54.377,-44.568,-178.913,5.422,148.618
C07981=1228.305,54.127,-44.551,-178.916,5.422,148.618
C07982=1228.310,53.878,-44.534,-178.918,5.421,148.619
C07983=1228.314,53.628,-44.517,-178.921,5.421,148.620
C07984=1228.320,53.379,-44.501,-178.924,5.420,148.620
C07985=1228.325,53.130,-44.484,-178.926,5.420,148.621
C07986=1228.329,52.880,-44.467,-178.929,5.419,148.622
C07987=1228.334,52.632,-44.451,-178.931,5.418,148.622
C07988=1228.339,52.382,-44.434,-178.934,5.417,148.623
C07989=1228.344,52.132,-44.417,-178.936,5.417,148.624
C07990=1228.349,51.884,-44.401,-178.939,5.416,148.624
C07991=1228.354,51.633,-44.384,-178.942,5.416,148.625
C07992=1228.359,51.384,-44.367,-178.944,5.415,148.626
C07993=1228.364,51.135,-44.351,-178.947,5.415,148.626
C07994=1228.369,50.885,-44.334,-178.950,5.414,148.627
C07995=1228.374,50.636,-44.317,-178.951,5.414,148.627
C07996=1228.379,50.387,-44.301,-178.954,5.413,148.628
C07997=1228.383,50.137,-44.284,-178.956,5.413,148.629
C07998=1228.388,49.887,-44.268,-178.959,5.412,148.629
C07999=1228.393,49.638,-44.252,-178.962,5.412,148.630
C08000=1228.398,49.389,-44.235,-178.964,5.411,148.631
C08001=1228.403,49.140,-44.218,-178.967,5.411,148.631
C08002=1228.408,48.890,-44.202,-178.970,5.410,148.632
C08003=1228.413,48.640,-44.186,-178.972,5.409,148.633
C08004=1228.419,48.391,-44.169,-178.974,5.408,148.633
C08005=1228.423,48.142,-44.152,-178.977,5.408,148.634
C08006=1228.428,47.892,-44.136,-178.980,5.407,148.635
C08007=1228.433,47.643,-44.120,-178.982,5.407,148.635
C08008=1228.437,47.393,-44.103,-178.984,5.407,148.636
C08009=1228.442,47.145,-44.087,-178.987,5.406,148.637
C08010=1228.448,46.895,-44.070,-178.990,5.406,148.637
C08011=1228.453,46.645,-44.054,-178.992,5.405,148.638
C08012=1228.458,46.396,-44.037,-178.995,5.405,148.639
C08013=1228.462,46.146,-44.021,-178.997,5.404,148.639
C08014=1228.467,45.897,-44.005,-179.000,5.403,148.640
C08015=1228.472,45.648,-43.989,-179.002,5.403,148.640
C08016=1228.477,45.399,-43.972,-179.005,5.402,148.641
C08017=1228.482,45.148,-43.956,-179.008,5.402,148.642
C08018=1228.488,44.900,-43.939,-179.010,5.401,148.642
C08019=1228.492,44.650,-43.923,-179.012,5.401,148.643
C08020=1228.497,44.401,-43.907,-179.015,5.401,148.644
C08021=1228.502,44.151,-43.890,-179.018,5.400,148.644
C08022=1228.506,43.902,-43.874,-179.020,5.400,148.645
C08023=1228.512,43.652,-43.858,-179.022,5.399,148.645
C08024=1228.516,43.403,-43.842,-179.025,5.398,148.646
C08025=1228.522,43.153,-43.826,-179.028,5.398,148.647
C08026=1228.526,42.904,-43.809,-179.030,5.397,148.647
C08027=1228.531,42.655,-43.793,-179.033,5.396,148.648
C08028=1228.536,42.405,-43.777,-179.035,5.397,148.649
C08029=1228.542,42.156,-43.760,-179.038,5.396,148.650
C08030=1228.547,41.906,-43.744,-179.040,5.396,148.650
C08031=1228.552,41.657,-43.728,-179.043,5.395,148.651
C08032=1228.556,41.407,-43.712,-179.046,5.394,148.652
C08033=1228.562,41.158,-43.696,-179.048,5.394,148.652
C08034=1228.566,40.909,-43.679,-179.050,5.393,148.653
C08035=1228.571,40.659,-43.663,-179.053,5.392,148.653
C08036=1228.576,40.410,-43.647,-179.056,5.392,148.654
C08037=1228.581,40.160,-43.631,-179.058,5.392,148.655
C08038=1228.586,39.911,-43.614,-179.060,5.392,148.655
C08039=1228.591,39.661,-43.599,-179.063,5.391,148.656
C08040=1228.596,39.411,-43.583,-179.066,5.390,148.657
C08041=1228.601,39.163,-43.567,-179.068,5.390,148.657
C08042=1228.606,38.913,-43.551,-179.071,5.389,148.658
C08043=1228.611,38.664,-43.534,-179.073,5.389,148.659
C08044=1228.616,38.414,-43.519,-179.076,5.388,148.659
C08045=1228.621,38.165,-43.502,-179.078,5.388,148.660
C08046=1228.626,37.915,-43.486,-179.080,5.387,148.661
C08047=1228.631,37.666,-43.470,-179.083,5.387,148.661
C08048=1228.636,37.417,-43.454,-179.086,5.386,148.662
C08049=1228.640,37.167,-43.439,-179.088,5.386,148.663
C08050=1228.645,36.918,-43.423,-179.091,5.385,148.663
C08051=1228.651,36.669,-43.407,-179.094,5.385,148.664
C08052=1228.655,36.419,-43.390,-179.096,5.384,148.665
C08053=1228.660,36.170,-43.375,-179.098,5.384,148.665
C08054=1228.665,35.920,-43.359,-179.101,5.384,148.666
C08055=1228.670,35.671,-43.342,-179.104,5.383,148.667
C08056=1228.676,35.421,-43.327,-179.106,5.383,148.667
C08057=1228.680,35.171,-43.311,-179.109,5.382,148.668
C08058=1228.686,34.923,-43.295,-179.111,5.382,148.669
C08059=1228.690,34.672,-43.279,-179.114,5.381,148.669
C08060=1228.695,34.423,-43.264,-179.116,5.381,148.670
C08061=1228.700,34.175,-43.247,-179.118,5.380,148.670
C08062=1228.705,33.924,-43.231,-179.121,5.380,148.671
C08063=1228.710,33.675,-43.216,-179.124,5.379,148.672
C08064=1228.715,33.425,-43.200,-179.126,5.379,148.672
C08065=1228.720,33.176,-43.184,-179.129,5.378,148.673
C08066=1228.725,32.927,-43.168,-179.132,5.378,148.674
C08067=1228.730,32.677,-43.153,-179.134,5.378,148.675
C08068=1228.735,32.428,-43.136,-179.136,5.377,148.675
C08069=1228.740,32.179,-43.121,-179.139,5.377,148.676
C08070=1228.745,31.929,-43.105,-179.142,5.376,148.677
C08071=1228.750,31.679,-43.089,-179.144,5.376,148.677
C08072=1228.754,31.429,-43.074,-179.147,5.375,148.678
C08073=1228.759,31.181,-43.058,-179.149,5.375,148.679
C08074=1228.765,30.931,-43.042,-179.151,5.374,148.679
C08075=1228.769,30.681,-43.026,-179.154,5.374,148.680
C08076=1228.775,30.432,-43.010,-179.156,5.373,148.680
C08077=1228.779,30.183,-42.995,-179.159,5.373,148.681
C08078=1228.785,29.914,-42.978,-179.162,5.372,148.682
C08079=1228.790,29.645,-42.961,-179.165,5.372,148.683
C08080=1228.796,29.377,-42.944,-179.167,5.372,148.683
C08081=1228.801,29.108,-42.927,-179.170,5.371,148.684
C08082=1228.806,28.859,-42.912,-179.173,5.370,148.685
C08083=1228.811,28.609,-42.896,-179.175,5.371,148.685
C08084=1228.816,28.359,-42.880,-179.177,5.370,148.686
C08085=1228.821,28.110,-42.865,-179.180,5.370,148.687
C08086=1228.826,27.862,-42.849,-179.183,5.369,148.687
C08087=1228.830,27.611,-42.833,-179.185,5.369,148.688
C08088=1228.836,27.362,-42.818,-179.188,5.368,148.689
C08089=1228.840,27.113,-42.803,-179.190,5.368,148.689
C08090=1228.845,26.863,-42.787,-179.193,5.368,148.690
C08091=1228.851,26.613,-42.771,-179.195,5.367,148.691
C08092=1228.856,26.364,-42.755,-179.197,5.366,148.691
C08093=1228.861,26.115,-42.740,-179.200,5.366,148.692
C08094=1228.865,25.865,-42.725,-179.202,5.366,148.693
C08095=1228.871,25.615,-42.709,-179.205,5.365,148.693
C08096=1228.876,25.366,-42.694,-179.208,5.365,148.694
C08097=1228.880,25.116,-42.678,-179.210,5.364,148.695
C08098=1228.886,24.867,-42.662,-179.213,5.364,148.695
C08099=1228.890,24.618,-42.647,-179.215,5.363,148.696
C08100=1228.896,24.368,-42.632,-179.218,5.363,148.697
C08101=1228.901,24.118,-42.616,-179.220,5.363,148.697
C08102=1228.905,23.869,-42.601,-179.223,5.362,148.698
C08103=1228.911,23.620,-42.585,-179.225,5.362,148.699
C08104=1228.915,23.371,-42.570,-179.228,5.361,148.699
C08105=1228.921,23.121,-42.555,-179.230,5.362,148.700
C08106=1228.925,22.871,-42.539,-179.233,5.361,148.701
C08107=1228.930,22.622,-42.524,-179.235,5.360,148.701
C08108=1228.935,22.373,-42.508,-179.238,5.360,148.702
C08109=1228.940,22.124,-42.493,-179.241,5.359,148.703
C08110=1228.945,21.874,-42.477,-179.243,5.359,148.703
C08111=1228.951,21.623,-42.462,-179.245,5.359,148.704
C08112=1228.955,21.374,-42.447,-179.248,5.359,148.705
C08113=1228.961,21.125,-42.432,-179.251,5.358,148.706
C08114=1228.965,20.876,-42.417,-179.253,5.357,148.706
C08115=1228.970,20.626,-42.401,-179.256,5.357,148.707
C08116=1228.975,20.377,-42.386,-179.258,5.357,148.707
C08117=1228.980,20.127,-42.370,-179.260,5.356,148.708
C08118=1228.985,19.878,-42.355,-179.263,5.356,148.709
C08119=1228.990,19.628,-42.340,-179.266,5.355,148.709
C08120=1228.996,19.379,-42.325,-179.268,5.355,148.710
C08121=1229.000,19.129,-42.309,-179.270,5.355,148.711
C08122=1229.005,18.880,-42.294,-179.273,5.354,148.711
C08123=1229.010,18.631,-42.279,-179.276,5.354,148.712
C08124=1229.016,18.380,-42.264,-179.278,5.353,148.713
C08125=1229.020,18.131,-42.249,-179.280,5.354,148.714
C08126=1229.026,17.882,-42.233,-179.283,5.353,148.714
C08127=1229.030,17.632,-42.218,-179.286,5.352,148.715
C08128=1229.035,17.383,-42.202,-179.288,5.352,148.716
C08129=1229.040,17.133,-42.188,-179.291,5.351,148.716
C08130=1229.045,16.884,-42.173,-179.293,5.352,148.717
C08131=1229.050,16.635,-42.158,-179.296,5.351,148.718
C08132=1229.055,16.385,-42.142,-179.298,5.351,148.718
C08133=1229.060,16.135,-42.128,-179.301,5.350,148.719
C08134=1229.066,15.886,-42.112,-179.304,5.350,148.720
C08135=1229.070,15.636,-42.097,-179.306,5.350,148.720
C08136=1229.075,15.387,-42.082,-179.308,5.349,148.721
C08137=1229.080,15.137,-42.067,-179.311,5.349,148.722
C08138=1229.085,14.888,-42.052,-179.314,5.348,148.722
C08139=1229.090,14.639,-42.036,-179.316,5.348,148.723
C08140=1229.095,14.389,-42.022,-179.318,5.348,148.724
C08141=1229.101,14.140,-42.006,-179.321,5.347,148.724
C08142=1229.105,13.890,-41.991,-179.324,5.347,148.725
C08143=1229.110,13.641,-41.977,-179.326,5.346,148.726
C08144=1229.115,13.391,-41.961,-179.328,5.347,148.726
C08145=1229.120,13.141,-41.947,-179.331,5.346,148.727
C08146=1229.125,12.892,-41.931,-179.334,5.346,148.728
C08147=1229.130,12.642,-41.916,-179.336,5.345,148.729
C08148=1229.135,12.393,-41.902,-179.338,5.345,148.729
C08149=1229.140,12.143,-41.887,-179.341,5.345,148.730
C08150=1229.145,11.894,-41.872,-179.344,5.344,148.731
C08151=1229.150,11.645,-41.857,-179.346,5.344,148.731
C08152=1229.155,11.395,-41.842,-179.348,5.344,148.732
C08153=1229.160,11.145,-41.827,-179.351,5.343,148.733
C08154=1229.165,10.896,-41.812,-179.354,5.343,148.733
C08155=1229.171,10.646,-41.798,-179.356,5.342,148.734
C08156=1229.175,10.397,-41.783,-179.359,5.342,148.735
C08157=1229.180,10.148,-41.768,-179.361,5.342,148.735
C08158=1229.185,9.898,-41.753,-179.364,5.342,148.736
C08159=1229.190,9.648,-41.738,-179.366,5.341,148.737
C08160=1229.195,9.399,-41.723,-179.369,5.340,148.737
C08161=1229.200,9.150,-41.708,-179.371,5.341,148.738
C08162=1229.205,8.900,-41.694,-179.374,5.340,148.739
C08163=1229.210,8.650,-41.679,-179.376,5.340,148.740
C08164=1229.216,8.401,-41.664,-179.379,5.339,148.740
C08165=1229.221,8.151,-41.649,-179.381,5.339,148.741
C08166=1229.225,7.902,-41.634,-179.384,5.339,148.742
C08167=1229.230,7.652,-41.620,-179.386,5.338,148.742
C08168=1229.235,7.402,-41.604,-179.389,5.338,148.743
C08169=1229.240,7.153,-41.590,-179.391,5.338,148.743
C08170=1229.245,6.904,-41.575,-179.393,5.337,148.744
C08171=1229.250,6.654,-41.561,-179.396,5.337,148.745
C08172=1229.256,6.405,-41.545,-179.399,5.336,148.745
C08173=1229.261,6.156,-41.531,-179.401,5.336,148.746
C08174=1229.266,5.906,-41.517,-179.403,5.336,148.747
C08175=1229.270,5.657,-41.502,-179.406,5.335,148.748
C08176=1229.276,5.407,-41.487,-179.409,5.335,148.748
C08177=1229.281,5.158,-41.472,-179.411,5.335,148.749
C08178=1229.286,4.908,-41.458,-179.413,5.335,148.750
C08179=1229.290,4.658,-41.443,-179.416,5.334,148.750
C08180=1229.295,4.409,-41.428,-179.419,5.334,148.751
C08181=1229.301,4.159,-41.414,-179.421,5.334,148.752
C08182=1229.306,3.890,-41.398,-179.424,5.334,148.753
C08183=1229.311,3.622,-41.382,-179.427,5.333,148.753
C08184=1229.316,3.353,-41.366,-179.429,5.333,148.754
C08185=1229.322,3.083,-41.351,-179.432,5.332,148.755
C08186=1229.327,2.834,-41.336,-179.434,5.332,148.755
C08187=1229.332,2.584,-41.322,-179.437,5.332,148.756
C08188=1229.337,2.334,-41.307,-179.439,5.331,148.757
C08189=1229.342,2.085,-41.292,-179.442,5.331,148.757
C08190=1229.347,1.835,-41.277,-179.444,5.331,148.758
C08191=1229.353,1.586,-41.264,-179.447,5.331,148.759
C08192=1229.358,1.337,-41.249,-179.449,5.330,148.759
C08193=1229.362,1.088,-41.234,-179.452,5.329,148.760
C08194=1229.367,0.838,-41.220,-179.454,5.330,148.761
C08195=1229.372,0.588,-41.206,-179.457,5.329,148.762
C08196=1229.377,0.338,-41.191,-179.459,5.329,148.762
C08197=1229.382,0.089,-41.176,-179.461,5.329,148.763
C08198=1229.388,-0.161,-41.162,-179.464,5.328,148.764
C08199=1229.393,-0.410,-41.147,-179.467,5.328,148.764
C08200=1229.398,-0.660,-41.133,-179.469,5.327,148.765
C08201=1229.403,-0.908,-41.118,-179.471,5.328,148.766
C08202=1229.408,-1.158,-41.104,-179.474,5.327,148.766
C08203=1229.413,-1.408,-41.090,-179.477,5.327,148.767
C08204=1229.418,-1.658,-41.076,-179.480,5.326,148.768
C08205=1229.423,-1.907,-41.061,-179.482,5.327,148.769
C08206=1229.428,-2.157,-41.047,-179.485,5.326,148.769
C08207=1229.432,-2.406,-41.032,-179.487,5.326,148.770
C08208=1229.438,-2.655,-41.018,-179.489,5.326,148.771
C08209=1229.443,-2.905,-41.004,-179.492,5.325,148.771
C08210=1229.448,-3.155,-40.990,-179.495,5.325,148.772
C08211=1229.453,-3.404,-40.975,-179.497,5.324,148.773
C08212=1229.458,-3.654,-40.961,-179.499,5.325,148.773
C08213=1229.463,-3.904,-40.947,-179.502,5.324,148.774
C08214=1229.468,-4.153,-40.932,-179.505,5.324,148.775
C08215=1229.473,-4.402,-40.919,-179.507,5.324,148.776
C08216=1229.478,-4.652,-40.904,-179.509,5.323,148.776
C08217=1229.483,-4.901,-40.889,-179.512,5.323,148.777
C08218=1229.488,-5.151,-40.875,-179.514,5.323,148.778
C08219=1229.493,-5.401,-40.861,-179.517,5.323,148.778
C08220=1229.498,-5.650,-40.847,-179.519,5.322,148.779
C08221=1229.503,-5.899,-40.832,-179.522,5.322,148.780
C08222=1229.508,-6.149,-40.818,-179.524,5.322,148.780
C08223=1229.513,-6.399,-40.804,-179.527,5.321,148.781
C08224=1229.518,-6.649,-40.790,-179.529,5.321,148.782
C08225=1229.524,-6.898,-40.776,-179.532,5.321,148.782
C08226=1229.528,-7.147,-40.761,-179.534,5.321,148.783
C08227=1229.533,-7.397,-40.747,-179.537,5.320,148.784
C08228=1229.538,-7.647,-40.733,-179.539,5.320,148.785
C08229=1229.543,-7.896,-40.719,-179.542,5.320,148.785
C08230=1229.549,-8.145,-40.705,-179.544,5.319,148.786
C08231=1229.554,-8.395,-40.690,-179.547,5.319,148.787
C08232=1229.559,-8.645,-40.676,-179.549,5.319,148.787
C08233=1229.564,-8.894,-40.662,-179.552,5.319,148.788
C08234=1229.569,-9.143,-40.649,-179.554,5.318,148.789
C08235=1229.574,-9.393,-40.634,-179.556,5.318,148.789
C08236=1229.578,-9.643,-40.620,-179.559,5.318,148.790
C08237=1229.584,-9.893,-40.606,-179.562,5.317,148.791
C08238=1229.589,-10.143,-40.592,-179.564,5.318,148.791
C08239=1229.594,-10.392,-40.578,-179.566,5.317,148.792
C08240=1229.599,-10.641,-40.564,-179.569,5.317,148.793
C08241=1229.604,-10.891,-40.550,-179.571,5.317,148.794
C08242=1229.610,-11.140,-40.536,-179.574,5.316,148.794
C08243=1229.614,-11.389,-40.522,-179.576,5.316,148.795
C08244=1229.619,-11.639,-40.508,-179.579,5.316,148.796
C08245=1229.624,-11.889,-40.494,-179.581,5.316,148.796
C08246=1229.630,-12.139,-40.480,-179.584,5.315,148.797
C08247=1229.635,-12.388,-40.466,-179.587,5.315,148.798
C08248=1229.640,-12.638,-40.452,-179.589,5.315,148.798
C08249=1229.644,-12.887,-40.438,-179.591,5.314,148.799
C08250=1229.649,-13.136,-40.424,-179.594,5.314,148.800
C08251=1229.654,-13.386,-40.410,-179.596,5.314,148.800
C08252=1229.660,-13.636,-40.396,-179.599,5.314,148.801
C08253=1229.665,-13.885,-40.382,-179.601,5.313,148.802
C08254=1229.669,-14.135,-40.369,-179.603,5.314,148.803
C08255=1229.674,-14.385,-40.355,-179.606,5.313,148.803
C08256=1229.680,-14.634,-40.341,-179.609,5.312,148.804
C08257=1229.685,-14.884,-40.327,-179.611,5.313,148.805
C08258=1229.690,-15.134,-40.313,-179.613,5.312,148.805
C08259=1229.695,-15.382,-40.299,-179.617,5.312,148.806
C08260=1229.700,-15.633,-40.286,-179.619,5.312,148.807
C08261=1229.705,-15.882,-40.272,-179.621,5.312,148.808
C08262=1229.711,-16.131,-40.258,-179.624,5.311,148.808
C08263=1229.715,-16.381,-40.244,-179.626,5.312,148.809
C08264=1229.720,-16.631,-40.230,-179.629,5.311,148.810
C08265=1229.726,-16.880,-40.217,-179.631,5.311,148.810
C08266=1229.731,-17.130,-40.202,-179.633,5.311,148.811
C08267=1229.735,-17.380,-40.189,-179.636,5.310,148.812
C08268=1229.741,-17.629,-40.175,-179.639,5.310,148.812
C08269=1229.746,-17.879,-40.161,-179.641,5.310,148.813
C08270=1229.751,-18.129,-40.148,-179.644,5.310,148.814
C08271=1229.756,-18.378,-40.134,-179.646,5.309,148.815
C08272=1229.761,-18.627,-40.120,-179.648,5.310,148.815
C08273=1229.767,-18.877,-40.107,-179.651,5.309,148.816
C08274=1229.771,-19.126,-40.093,-179.654,5.309,148.817
C08275=1229.776,-19.376,-40.079,-179.656,5.309,148.817
C08276=1229.782,-19.626,-40.066,-179.658,5.308,148.818
C08277=1229.786,-19.875,-40.052,-179.661,5.308,148.819
C08278=1229.791,-20.125,-40.038,-179.663,5.308,148.819
C08279=1229.797,-20.374,-40.024,-179.666,5.308,148.820
C08280=1229.801,-20.624,-40.011,-179.668,5.307,148.821
C08281=1229.807,-20.873,-39.998,-179.670,5.307,148.822
C08282=1229.812,-21.123,-39.983,-179.673,5.307,148.822
C08283=1229.816,-21.373,-39.970,-179.676,5.306,148.823
C08284=1229.822,-21.622,-39.956,-179.678,5.307,148.824
C08285=1229.827,-21.872,-39.942,-179.681,5.306,148.824
C08286=1229.832,-22.141,-39.929,-179.684,5.306,148.825
C08287=1229.838,-22.410,-39.914,-179.686,5.306,148.826
C08288=1229.843,-22.680,-39.899,-179.688,5.306,148.827
C08289=1229.849,-22.949,-39.884,-179.691,5.305,148.827
C08290=1229.854,-23.198,-39.871,-179.694,5.305,148.828
C08291=1229.859,-23.448,-39.857,-179.696,5.305,148.829
C08292=1229.865,-23.698,-39.844,-179.698,5.305,148.829
C08293=1229.869,-23.947,-39.830,-179.701,5.304,148.830
C08294=1229.875,-24.197,-39.817,-179.703,5.304,148.831
C08295=1229.879,-24.446,-39.803,-179.706,5.304,148.832
C08296=1229.884,-24.697,-39.790,-179.708,5.305,148.832
C08297=1229.889,-24.945,-39.776,-179.711,5.304,148.833
C08298=1229.894,-25.196,-39.763,-179.714,5.304,148.834
C08299=1229.899,-25.444,-39.749,-179.716,5.304,148.835
C08300=1229.904,-25.695,-39.736,-179.719,5.303,148.835
C08301=1229.910,-25.944,-39.722,-179.721,5.303,148.836
C08302=1229.914,-26.194,-39.709,-179.723,5.303,148.837
C08303=1229.920,-26.443,-39.696,-179.726,5.303,148.837
C08304=1229.924,-26.693,-39.682,-179.729,5.302,148.838
C08305=1229.930,-26.942,-39.669,-179.731,5.302,148.839
C08306=1229.935,-27.192,-39.655,-179.733,5.302,148.839
C08307=1229.940,-27.441,-39.642,-179.735,5.302,148.840
C08308=1229.945,-27.691,-39.629,-179.738,5.302,148.841
C08309=1229.950,-27.940,-39.615,-179.741,5.301,148.841
C08310=1229.955,-28.190,-39.602,-179.743,5.302,148.842
C08311=1229.961,-28.439,-39.588,-179.745,5.301,148.843
C08312=1229.965,-28.689,-39.575,-179.748,5.301,148.844
C08313=1229.971,-28.939,-39.562,-179.750,5.301,148.844
C08314=1229.975,-29.188,-39.548,-179.753,5.300,148.845
C08315=1229.981,-29.438,-39.535,-179.756,5.300,148.846
C08316=1229.986,-29.688,-39.522,-179.758,5.300,148.846
C08317=1229.991,-29.937,-39.508,-179.760,5.300,148.847
C08318=1229.996,-30.187,-39.495,-179.762,5.300,148.848
C08319=1230.001,-30.436,-39.483,-179.765,5.299,148.848
C08320=1230.006,-30.687,-39.469,-179.768,5.299,148.849
C08321=1230.011,-30.935,-39.456,-179.770,5.299,148.850
C08322=1230.016,-31.186,-39.442,-179.772,5.299,148.851
C08323=1230.021,-31.435,-39.430,-179.775,5.298,148.851
C08324=1230.027,-31.684,-39.416,-179.777,5.299,148.852
C08325=1230.031,-31.934,-39.403,-179.780,5.298,148.853
C08326=1230.036,-32.183,-39.390,-179.782,5.299,148.854
C08327=1230.042,-32.434,-39.377,-179.785,5.298,148.854
C08328=1230.046,-32.682,-39.363,-179.788,5.298,148.855
C08329=1230.052,-32.933,-39.350,-179.790,5.298,148.856
C08330=1230.057,-33.182,-39.337,-179.792,5.298,148.856
C08331=1230.062,-33.431,-39.325,-179.795,5.298,148.857
C08332=1230.067,-33.682,-39.311,-179.797,5.297,148.858
C08333=1230.072,-33.930,-39.298,-179.800,5.297,148.858
C08334=1230.077,-34.181,-39.284,-179.802,5.297,148.859
C08335=1230.082,-34.430,-39.272,-179.805,5.297,148.860
C08336=1230.087,-34.680,-39.259,-179.807,5.296,148.861
C08337=1230.093,-34.930,-39.245,-179.809,5.297,148.861
C08338=1230.098,-35.179,-39.233,-179.812,5.296,148.862
C08339=1230.102,-35.428,-39.219,-179.814,5.296,148.863
C08340=1230.108,-35.678,-39.206,-179.817,5.296,148.863
C08341=1230.113,-35.927,-39.193,-179.819,5.295,148.864
C08342=1230.118,-36.177,-39.180,-179.822,5.296,148.865
C08343=1230.124,-36.427,-39.167,-179.824,5.295,148.865
C08344=1230.128,-36.677,-39.154,-179.826,5.296,148.866
C08345=1230.133,-36.926,-39.142,-179.829,5.295,148.867
C08346=1230.139,-37.176,-39.128,-179.832,5.295,148.868
C08347=1230.143,-37.425,-39.115,-179.834,5.295,148.868
C08348=1230.148,-37.675,-39.102,-179.836,5.294,148.869
C08349=1230.154,-37.924,-39.089,-179.838,5.295,148.870
C08350=1230.159,-38.174,-39.076,-179.841,5.294,148.870
C08351=1230.164,-38.424,-39.063,-179.844,5.294,148.871
C08352=1230.169,-38.673,-39.051,-179.846,5.294,148.872
C08353=1230.174,-38.923,-39.037,-179.849,5.294,148.873
C08354=1230.179,-39.173,-39.025,-179.851,5.294,148.873
C08355=1230.185,-39.422,-39.012,-179.854,5.294,148.874
C08356=1230.190,-39.672,-38.998,-179.856,5.293,148.875
C08357=1230.195,-39.922,-38.986,-179.859,5.294,148.876
C08358=1230.200,-40.171,-38.973,-179.861,5.293,148.876
C08359=1230.205,-40.421,-38.960,-179.863,5.293,148.877
C08360=1230.210,-40.671,-38.947,-179.866,5.293,148.878
C08361=1230.216,-40.920,-38.935,-179.869,5.292,148.878
C08362=1230.220,-41.170,-38.922,-179.871,5.293,148.879
C08363=1230.225,-41.419,-38.909,-179.873,5.292,148.880
C08364=1230.230,-41.669,-38.896,-179.875,5.293,148.880
C08365=1230.236,-41.919,-38.883,-179.878,5.292,148.881
C08366=1230.241,-42.168,-38.870,-179.881,5.292,148.882
C08367=1230.246,-42.418,-38.858,-179.883,5.292,148.883
C08368=1230.250,-42.668,-38.845,-179.885,5.291,148.883
C08369=1230.255,-42.917,-38.832,-179.888,5.292,148.884
C08370=1230.261,-43.166,-38.819,-179.890,5.291,148.885
C08371=1230.266,-43.416,-38.806,-179.893,5.291,148.885
C08372=1230.271,-43.666,-38.793,-179.895,5.291,148.886
C08373=1230.276,-43.916,-38.781,-179.898,5.291,148.887
C08374=1230.282,-44.165,-38.769,-179.900,5.291,148.887
C08375=1230.286,-44.415,-38.756,-179.902,5.290,148.888
C08376=1230.292,-44.665,-38.743,-179.904,5.291,148.889
C08377=1230.297,-44.914,-38.730,-179.907,5.290,148.890
C08378=1230.302,-45.163,-38.717,-179.910,5.290,148.890
C08379=1230.307,-45.413,-38.704,-179.912,5.290,148.891
C08380=1230.312,-45.663,-38.692,-179.915,5.290,148.892
C08381=1230.317,-45.913,-38.680,-179.917,5.290,148.893
C08382=1230.322,-46.162,-38.667,-179.920,5.290,148.893
C08383=1230.327,-46.412,-38.654,-179.922,5.289,148.894
C08384=1230.333,-46.662,-38.641,-179.925,5.290,148.895
C08385=1230.338,-46.911,-38.629,-179.927,5.289,148.895
C08386=1230.343,-47.160,-38.616,-179.929,5.289,148.896
C08387=1230.348,-47.410,-38.604,-179.932,5.289,148.897
C08388=1230.353,-47.660,-38.591,-179.934,5.289,148.897
C08389=1230.358,-47.909,-38.579,-179.937,5.289,148.898
C08390=1230.363,-48.179,-38.565,-179.939,5.288,148.899
C08391=1230.370,-48.449,-38.552,-179.941,5.289,148.900
C08392=1230.375,-48.719,-38.538,-179.945,5.289,148.901
C08393=1230.380,-48.989,-38.524,-179.947,5.288,148.901
C08394=1230.385,-49.238,-38.512,-179.949,5.288,148.902
C08395=1230.391,-49.488,-38.499,-179.952,5.288,148.903
C08396=1230.396,-49.738,-38.487,-179.955,5.287,148.903
C08397=1230.401,-49.987,-38.474,-179.957,5.288,148.904
C08398=1230.406,-50.237,-38.461,-179.959,5.287,148.905
C08399=1230.411,-50.487,-38.449,-179.962,5.288,148.905
C08400=1230.416,-50.736,-38.437,-179.964,5.287,148.906
C08401=1230.421,-50.985,-38.424,-179.966,5.287,148.907
C08402=1230.427,-51.235,-38.412,-179.969,5.287,148.908
C08403=1230.432,-51.485,-38.399,-179.972,5.286,148.908
C08404=1230.437,-51.735,-38.387,-179.974,5.287,148.909
C08405=1230.442,-51.985,-38.375,-179.976,5.286,148.910
C08406=1230.447,-52.234,-38.362,-179.978,5.287,148.910
C08407=1230.452,-52.483,-38.349,-179.981,5.286,148.911
C08408=1230.458,-52.733,-38.338,-179.983,5.286,148.912
C08409=1230.463,-52.983,-38.325,-179.986,5.286,148.912
C08410=1230.467,-53.233,-38.312,-179.989,5.285,148.913
C08411=1230.473,-53.482,-38.300,-179.991,5.286,148.914
C08412=1230.478,-53.732,-38.287,-179.994,5.286,148.915
C08413=1230.483,-53.981,-38.275,-179.996,5.286,148.916
C08414=1230.488,-54.231,-38.264,-179.999,5.286,148.916
C08415=1230.493,-54.480,-38.251,179.999,5.286,148.917
C08416=1230.498,-54.730,-38.239,179.997,5.285,148.918
C08417=1230.503,-54.980,-38.226,179.995,5.286,148.918
C08418=1230.508,-55.229,-38.214,179.992,5.285,148.919
C08419=1230.513,-55.479,-38.202,179.989,5.285,148.920
C08420=1230.518,-55.729,-38.189,179.987,5.285,148.920
C08421=1230.524,-55.979,-38.177,179.984,5.285,148.921
C08422=1230.529,-56.228,-38.165,179.982,5.285,148.922
C08423=1230.534,-56.478,-38.153,179.980,5.284,148.923
C08424=1230.540,-56.727,-38.140,179.978,5.285,148.923
C08425=1230.544,-56.978,-38.128,179.975,5.284,148.924
C08426=1230.549,-57.227,-38.116,179.973,5.285,148.925
C08427=1230.554,-57.477,-38.104,179.970,5.284,148.925
C08428=1230.559,-57.726,-38.091,179.968,5.284,148.926
C08429=1230.565,-57.976,-38.079,179.965,5.284,148.927
C08430=1230.570,-58.225,-38.067,179.963,5.284,148.927
C08431=1230.575,-58.475,-38.055,179.961,5.284,148.928
C08432=1230.580,-58.725,-38.042,179.958,5.283,148.929
C08433=1230.585,-58.974,-38.031,179.956,5.284,148.930
C08434=1230.590,-59.223,-38.018,179.953,5.283,148.930
C08435=1230.596,-59.473,-38.007,179.951,5.284,148.931
C08436=1230.601,-59.723,-37.994,179.949,5.283,148.932
C08437=1230.606,-59.973,-37.982,179.946,5.283,148.932
C08438=1230.611,-60.223,-37.969,179.944,5.283,148.933
C08439=1230.616,-60.473,-37.957,179.941,5.282,148.934
C08440=1230.621,-60.722,-37.946,179.939,5.283,148.935
C08441=1230.626,-60.972,-37.933,179.936,5.282,148.935
C08442=1230.631,-61.221,-37.921,179.934,5.283,148.936
C08443=1230.637,-61.471,-37.909,179.932,5.282,148.937
C08444=1230.642,-61.721,-37.897,179.930,5.283,148.937
C08445=1230.647,-61.970,-37.886,179.927,5.282,148.938
C08446=1230.652,-62.220,-37.873,179.925,5.282,148.939
C08447=1230.657,-62.470,-37.861,179.922,5.282,148.939
C08448=1230.662,-62.719,-37.849,179.920,5.282,148.940
C08449=1230.667,-62.969,-37.837,179.917,5.282,148.941
C08450=1230.672,-63.218,-37.825,179.914,5.282,148.942
C08451=1230.678,-63.468,-37.813,179.912,5.282,148.943
C08452=1230.683,-63.718,-37.801,179.909,5.282,148.943
C08453=1230.688,-63.968,-37.789,179.907,5.282,148.944
C08454=1230.693,-64.217,-37.777,179.905,5.281,148.945
C08455=1230.698,-64.467,-37.765,179.903,5.282,148.945
C08456=1230.704,-64.717,-37.753,179.900,5.281,148.946
C08457=1230.708,-64.966,-37.741,179.898,5.282,148.947
C08458=1230.713,-65.216,-37.729,179.895,5.281,148.947
C08459=1230.719,-65.465,-37.718,179.893,5.281,148.948
C08460=1230.724,-65.715,-37.706,179.890,5.281,148.949
C08461=1230.729,-65.964,-37.694,179.888,5.281,148.950
C08462=1230.734,-66.214,-37.682,179.886,5.281,148.950
C08463=1230.740,-66.464,-37.670,179.883,5.280,148.951
C08464=1230.744,-66.714,-37.659,179.881,5.281,148.952
C08465=1230.749,-66.963,-37.646,179.878,5.280,148.952
C08466=1230.755,-67.213,-37.634,179.876,5.281,148.953
C08467=1230.760,-67.463,-37.622,179.873,5.280,148.954
C08468=1230.765,-67.713,-37.611,179.871,5.280,148.955
C08469=1230.770,-67.962,-37.598,179.869,5.280,148.955
C08470=1230.776,-68.212,-37.586,179.867,5.280,148.956
C08471=1230.781,-68.461,-37.576,179.864,5.280,148.957
C08472=1230.786,-68.711,-37.564,179.862,5.280,148.957
C08473=1230.792,-68.961,-37.552,179.859,5.280,148.958
C08474=1230.796,-69.210,-37.540,179.857,5.280,148.959
C08475=1230.801,-69.460,-37.528,179.854,5.280,148.960
C08476=1230.807,-69.710,-37.516,179.852,5.280,148.960
C08477=1230.812,-69.959,-37.505,179.850,5.279,148.961
C08478=1230.817,-70.209,-37.493,179.848,5.280,148.962
C08479=1230.822,-70.459,-37.481,179.845,5.279,148.962
C08480=1230.827,-70.709,-37.470,179.842,5.279,148.963
C08481=1230.832,-70.958,-37.457,179.840,5.279,148.964
C08482=1230.837,-71.208,-37.446,179.837,5.279,148.964
C08483=1230.843,-71.457,-37.434,179.835,5.279,148.965
C08484=1230.848,-71.707,-37.423,179.833,5.279,148.966
C08485=1230.853,-71.956,-37.411,179.831,5.279,148.967
C08486=1230.859,-72.206,-37.399,179.828,5.279,148.967
C08487=1230.863,-72.456,-37.388,179.826,5.279,148.968
C08488=1230.869,-72.706,-37.376,179.823,5.278,148.969
C08489=1230.873,-72.956,-37.365,179.821,5.279,148.969
C08490=1230.879,-73.206,-37.353,179.818,5.278,148.970
C08491=1230.884,-73.456,-37.341,179.816,5.279,148.971
C08492=1230.889,-73.704,-37.329,179.814,5.278,148.972
C08493=1230.895,-73.954,-37.317,179.812,5.278,148.972
C08494=1230.900,-74.225,-37.305,179.809,5.278,148.973
C08495=1230.906,-74.495,-37.292,179.806,5.278,148.974
C08496=1230.912,-74.765,-37.280,179.804,5.278,148.975
C08497=1230.917,-75.036,-37.267,179.801,5.278,148.975
C08498=1230.922,-75.285,-37.256,179.799,5.278,148.976
C08499=1230.928,-75.535,-37.245,179.796,5.278,148.977
C08500=1230.932,-75.784,-37.233,179.794,5.278,148.977
C08501=1230.938,-76.034,-37.221,179.791,5.278,148.978
C08502=1230.943,-76.284,-37.210,179.789,5.278,148.979
C08503=1230.948,-76.534,-37.198,179.787,5.277,148.980
C08504=1230.953,-76.783,-37.187,179.785,5.278,148.980
C08505=1230.959,-77.033,-37.175,179.782,5.277,148.981
C08506=1230.963,-77.282,-37.164,179.779,5.277,148.982
C08507=1230.969,-77.532,-37.152,179.777,5.277,148.982
C08508=1230.974,-77.782,-37.141,179.774,5.277,148.983
C08509=1230.979,-78.032,-37.129,179.772,5.277,148.984
C08510=1230.984,-78.281,-37.118,179.770,5.277,148.985
C08511=1230.989,-78.530,-37.107,179.768,5.277,148.985
C08512=1230.995,-78.781,-37.096,179.765,5.277,148.986
C08513=1230.999,-79.030,-37.084,179.763,5.277,148.987
C08514=1231.005,-79.280,-37.072,179.760,5.276,148.987
C08515=1231.010,-79.530,-37.061,179.758,5.277,148.988
C08516=1231.016,-79.779,-37.050,179.755,5.276,148.989
C08517=1231.020,-80.029,-37.038,179.753,5.277,148.989
C08518=1231.026,-80.279,-37.026,179.751,5.276,148.990
C08519=1231.030,-80.528,-37.015,179.749,5.277,148.991
C08520=1231.036,-80.777,-37.004,179.746,5.276,148.992
C08521=1231.041,-81.028,-36.993,179.744,5.276,148.992
C08522=1231.046,-81.277,-36.982,179.741,5.276,148.993
C08523=1231.052,-81.527,-36.970,179.739,5.276,148.994
C08524=1231.056,-81.777,-36.959,179.736,5.276,148.994
C08525=1231.062,-82.026,-36.948,179.734,5.276,148.995
C08526=1231.067,-82.276,-36.936,179.732,5.276,148.996
C08527=1231.072,-82.526,-36.925,179.730,5.276,148.997
C08528=1231.077,-82.776,-36.913,179.727,5.276,148.997
C08529=1231.083,-83.025,-36.902,179.725,5.276,148.998
C08530=1231.087,-83.275,-36.891,179.722,5.276,148.999
C08531=1231.093,-83.525,-36.880,179.720,5.276,148.999
C08532=1231.098,-83.775,-36.869,179.717,5.275,149.000
C08533=1231.103,-84.024,-36.858,179.715,5.276,149.001
C08534=1231.109,-84.274,-36.846,179.713,5.275,149.002
C08535=1231.113,-84.523,-36.835,179.710,5.276,149.002
C08536=1231.118,-84.774,-36.824,179.708,5.275,149.003
C08537=1231.124,-85.023,-36.812,179.706,5.276,149.004
C08538=1231.129,-85.272,-36.801,179.703,5.275,149.004
C08539=1231.134,-85.523,-36.791,179.701,5.275,149.005
C08540=1231.140,-85.772,-36.779,179.698,5.275,149.006
C08541=1231.145,-86.022,-36.768,179.696,5.275,149.007
C08542=1231.149,-86.271,-36.756,179.694,5.275,149.007
C08543=1231.154,-86.521,-36.746,179.691,5.275,149.008
C08544=1231.160,-86.771,-36.734,179.689,5.275,149.009
C08545=1231.165,-87.020,-36.723,179.687,5.275,149.009
C08546=1231.170,-87.271,-36.713,179.684,5.275,149.010
C08547=1231.176,-87.520,-36.701,179.682,5.275,149.011
C08548=1231.181,-87.769,-36.690,179.679,5.275,149.012
C08549=1231.186,-88.020,-36.679,179.677,5.275,149.012
C08550=1231.191,-88.269,-36.668,179.674,5.274,149.013
C08551=1231.196,-88.518,-36.656,179.672,5.275,149.014
C08552=1231.201,-88.769,-36.646,179.670,5.274,149.014
C08553=1231.207,-89.018,-36.635,179.668,5.275,149.015
C08554=1231.211,-89.267,-36.624,179.666,5.275,149.016
C08555=1231.217,-89.518,-36.612,179.663,5.275,149.016
C08556=1231.223,-89.767,-36.601,179.661,5.275,149.017
C08557=1231.228,-90.017,-36.591,179.658,5.275,149.018
C08558=1231.232,-90.267,-36.580,179.656,5.275,149.019
C08559=1231.238,-90.516,-36.568,179.653,5.274,149.019
C08560=1231.243,-90.766,-36.558,179.651,5.275,149.020
C08561=1231.248,-91.016,-36.546,179.649,5.274,149.021
C08562=1231.254,-91.265,-36.536,179.647,5.274,149.021
C08563=1231.258,-91.515,-36.525,179.644,5.274,149.022
C08564=1231.265,-91.765,-36.514,179.642,5.274,149.023
C08565=1231.269,-92.014,-36.503,179.639,5.274,149.023
C08566=1231.274,-92.265,-36.492,179.637,5.274,149.024
C08567=1231.280,-92.514,-36.481,179.635,5.274,149.025
C08568=1231.284,-92.763,-36.470,179.633,5.274,149.026
C08569=1231.290,-93.014,-36.459,179.630,5.274,149.026
C08570=1231.295,-93.263,-36.448,179.628,5.274,149.027
C08571=1231.300,-93.513,-36.437,179.625,5.274,149.028
C08572=1231.306,-93.762,-36.426,179.623,5.274,149.028
C08573=1231.311,-94.012,-36.416,179.620,5.273,149.029
C08574=1231.315,-94.262,-36.404,179.618,5.274,149.030
C08575=1231.322,-94.512,-36.394,179.616,5.273,149.030
C08576=1231.327,-94.762,-36.383,179.614,5.274,149.031
C08577=1231.332,-95.011,-36.372,179.611,5.273,149.032
C08578=1231.337,-95.261,-36.361,179.609,5.274,149.033
C08579=1231.342,-95.511,-36.350,179.606,5.273,149.033
C08580=1231.347,-95.760,-36.340,179.604,5.273,149.034
C08581=1231.352,-96.010,-36.329,179.601,5.273,149.035
C08582=1231.357,-96.259,-36.319,179.599,5.273,149.035
C08583=1231.363,-96.509,-36.307,179.597,5.273,149.036
C08584=1231.368,-96.759,-36.296,179.594,5.273,149.037
C08585=1231.373,-97.009,-36.286,179.592,5.274,149.038
C08586=1231.379,-97.258,-36.275,179.590,5.273,149.038
C08587=1231.384,-97.508,-36.264,179.588,5.274,149.039
C08588=1231.388,-97.758,-36.253,179.585,5.273,149.040
C08589=1231.394,-98.007,-36.243,179.583,5.273,149.040
C08590=1231.399,-98.258,-36.232,179.581,5.273,149.041
C08591=1231.404,-98.507,-36.221,179.579,5.273,149.042
C08592=1231.409,-98.757,-36.211,179.576,5.273,149.042
C08593=1231.415,-99.006,-36.201,179.574,5.273,149.043
C08594=1231.420,-99.256,-36.189,179.571,5.273,149.044
C08595=1231.425,-99.505,-36.179,179.569,5.273,149.045
C08596=1231.430,-99.756,-36.168,179.566,5.272,149.045
C08597=1231.435,-100.005,-36.158,179.564,5.273,149.046
C08598=1231.441,-100.276,-36.146,179.562,5.272,149.047
C08599=1231.447,-100.547,-36.134,179.559,5.273,149.048
C08600=1231.453,-100.818,-36.123,179.556,5.273,149.048
C08601=1231.458,-101.089,-36.111,179.554,5.272,149.049
C08602=1231.463,-101.339,-36.100,179.552,5.273,149.050
C08603=1231.469,-101.589,-36.090,179.549,5.273,149.050
C08604=1231.474,-101.838,-36.079,179.547,5.272,149.051
C08605=1231.479,-102.088,-36.069,179.545,5.273,149.052
C08606=1231.484,-102.338,-36.058,179.542,5.272,149.053
C08607=1231.490,-102.588,-36.048,179.540,5.273,149.053
C08608=1231.495,-102.837,-36.037,179.537,5.272,149.054
C08609=1231.500,-103.087,-36.026,179.536,5.272,149.055
C08610=1231.505,-103.337,-36.016,179.533,5.272,149.055
C08611=1231.511,-103.587,-36.006,179.531,5.272,149.056
C08612=1231.515,-103.836,-35.994,179.528,5.272,149.057
C08613=1231.520,-104.085,-35.985,179.526,5.272,149.057
C08614=1231.525,-104.336,-35.974,179.523,5.272,149.058
C08615=1231.531,-104.585,-35.964,179.521,5.272,149.059
C08616=1231.537,-104.835,-35.954,179.519,5.272,149.060
C08617=1231.541,-105.084,-35.942,179.517,5.272,149.060
C08618=1231.547,-105.334,-35.932,179.514,5.272,149.061
C08619=1231.552,-105.584,-35.922,179.512,5.272,149.062
C08620=1231.557,-105.834,-35.911,179.510,5.272,149.062
C08621=1231.562,-106.084,-35.901,179.507,5.272,149.063
C08622=1231.568,-106.333,-35.890,179.505,5.272,149.064
C08623=1231.573,-106.583,-35.879,179.502,5.272,149.065
C08624=1231.578,-106.833,-35.869,179.501,5.272,149.065
C08625=1231.584,-107.082,-35.859,179.498,5.271,149.066
C08626=1231.588,-107.332,-35.849,179.496,5.272,149.066
C08627=1231.594,-107.582,-35.839,179.493,5.271,149.067
C08628=1231.599,-107.832,-35.828,179.491,5.272,149.068
C08629=1231.604,-108.081,-35.818,179.488,5.271,149.069
C08630=1231.609,-108.331,-35.807,179.486,5.272,149.069
C08631=1231.615,-108.581,-35.796,179.484,5.271,149.070
C08632=1231.620,-108.830,-35.786,179.482,5.271,149.071
C08633=1231.625,-109.080,-35.776,179.479,5.272,149.071
C08634=1231.630,-109.330,-35.766,179.477,5.271,149.072
C08635=1231.635,-109.580,-35.755,179.475,5.272,149.073
C08636=1231.641,-109.829,-35.745,179.472,5.271,149.074
C08637=1231.646,-110.079,-35.735,179.470,5.272,149.074
C08638=1231.651,-110.329,-35.724,179.468,5.271,149.075
C08639=1231.657,-110.579,-35.714,179.466,5.271,149.075
C08640=1231.662,-110.828,-35.705,179.463,5.271,149.076
C08641=1231.667,-111.078,-35.694,179.461,5.271,149.077
C08642=1231.672,-111.328,-35.684,179.458,5.271,149.078
C08643=1231.677,-111.578,-35.673,179.456,5.271,149.078
C08644=1231.683,-111.828,-35.663,179.454,5.272,149.079
C08645=1231.688,-112.077,-35.653,179.451,5.271,149.080
C08646=1231.693,-112.327,-35.643,179.449,5.271,149.080
C08647=1231.698,-112.577,-35.633,179.447,5.271,149.081
C08648=1231.704,-112.826,-35.623,179.444,5.271,149.082
C08649=1231.709,-113.076,-35.612,179.442,5.271,149.082
C08650=1231.714,-113.326,-35.602,179.440,5.271,149.083
C08651=1231.719,-113.575,-35.592,179.438,5.270,149.084
C08652=1231.724,-113.825,-35.582,179.435,5.271,149.085
C08653=1231.730,-114.075,-35.571,179.433,5.270,149.085
C08654=1231.735,-114.324,-35.562,179.431,5.271,149.086
C08655=1231.740,-114.574,-35.551,179.429,5.271,149.087
C08656=1231.746,-114.824,-35.541,179.426,5.271,149.087
C08657=1231.751,-115.073,-35.531,179.424,5.271,149.088
C08658=1231.755,-115.323,-35.521,179.421,5.271,149.089
C08659=1231.761,-115.573,-35.511,179.419,5.271,149.090
C08660=1231.767,-115.823,-35.501,179.417,5.270,149.090
C08661=1231.772,-116.073,-35.490,179.415,5.271,149.091
C08662=1231.777,-116.323,-35.481,179.412,5.270,149.091
C08663=1231.782,-116.572,-35.471,179.410,5.271,149.092
C08664=1231.787,-116.822,-35.460,179.407,5.270,149.093
C08665=1231.792,-117.072,-35.450,179.405,5.270,149.094
C08666=1231.798,-117.321,-35.440,179.403,5.271,149.094
C08667=1231.803,-117.571,-35.430,179.400,5.270,149.095
C08668=1231.809,-117.822,-35.420,179.398,5.271,149.096
C08669=1231.814,-118.071,-35.411,179.396,5.270,149.096
C08670=1231.819,-118.320,-35.400,179.394,5.270,149.097
C08671=1231.824,-118.571,-35.390,179.391,5.270,149.098
C08672=1231.829,-118.820,-35.380,179.389,5.270,149.098
C08673=1231.835,-119.069,-35.370,179.387,5.270,149.099
C08674=1231.841,-119.320,-35.360,179.384,5.270,149.100
C08675=1231.845,-119.569,-35.350,179.382,5.270,149.101
C08676=1231.850,-119.819,-35.340,179.380,5.270,149.101
C08677=1231.855,-120.068,-35.331,179.378,5.271,149.102
C08678=1231.860,-120.318,-35.320,179.375,5.270,149.102
C08679=1231.866,-120.569,-35.311,179.373,5.270,149.103
C08680=1231.871,-120.818,-35.301,179.371,5.270,149.104
C08681=1231.877,-121.067,-35.291,179.369,5.270,149.105
C08682=1231.882,-121.318,-35.280,179.366,5.270,149.105
C08683=1231.887,-121.568,-35.271,179.364,5.270,149.106
C08684=1231.892,-121.817,-35.261,179.361,5.270,149.107
C08685=1231.897,-122.066,-35.251,179.359,5.270,149.107
C08686=1231.903,-122.316,-35.241,179.357,5.270,149.108
C08687=1231.908,-122.567,-35.231,179.355,5.270,149.109
C08688=1231.913,-122.816,-35.222,179.353,5.270,149.109
C08689=1231.919,-123.065,-35.212,179.350,5.269,149.110
C08690=1231.924,-123.315,-35.203,179.348,5.270,149.111
C08691=1231.929,-123.566,-35.192,179.345,5.269,149.112
C08692=1231.934,-123.815,-35.182,179.343,5.270,149.112
C08693=1231.940,-124.065,-35.173,179.340,5.269,149.113
C08694=1231.945,-124.314,-35.163,179.338,5.270,149.114
C08695=1231.950,-124.564,-35.153,179.337,5.270,149.114
C08696=1231.955,-124.815,-35.143,179.334,5.269,149.115
C08697=1231.960,-125.064,-35.134,179.332,5.270,149.116
C08698=1231.966,-125.313,-35.124,179.329,5.269,149.116
C08699=1231.971,-125.563,-35.115,179.327,5.270,149.117
C08700=1231.977,-125.813,-35.104,179.324,5.269,149.118
C08701=1231.982,-126.063,-35.094,179.322,5.270,149.119
C08702=1231.560,-126.074,-35.130,179.318,5.273,149.120
C08703=1231.555,-125.824,-35.139,179.321,5.272,149.120
C08704=1231.550,-125.574,-35.150,179.323,5.273,149.119
C08705=1231.544,-125.324,-35.160,179.325,5.273,149.118
C08706=1231.539,-125.074,-35.169,179.327,5.273,149.118
C08707=1231.533,-124.825,-35.179,179.330,5.273,149.117
C08708=1231.528,-124.575,-35.189,179.332,5.273,149.116
C08709=1231.523,-124.325,-35.198,179.334,5.273,149.116
C08710=1231.518,-124.075,-35.208,179.336,5.273,149.115
C08711=1231.513,-123.826,-35.218,179.339,5.273,149.114
C08712=1231.507,-123.576,-35.227,179.341,5.273,149.114
C08713=1231.502,-123.326,-35.237,179.343,5.273,149.113
C08714=1231.497,-123.076,-35.248,179.345,5.273,149.112
C08715=1231.492,-122.826,-35.257,179.348,5.273,149.112
C08716=1231.486,-122.577,-35.267,179.350,5.273,149.111
C08717=1231.481,-122.328,-35.277,179.353,5.273,149.110
C08718=1231.476,-122.077,-35.287,179.355,5.273,149.109
C08719=1231.470,-121.827,-35.297,179.357,5.273,149.109
C08720=1231.465,-121.578,-35.306,179.359,5.274,149.108
C08721=1231.460,-121.328,-35.317,179.361,5.273,149.107
C08722=1231.455,-121.079,-35.325,179.364,5.274,149.107
C08723=1231.450,-120.828,-35.336,179.366,5.273,149.106
C08724=1231.444,-120.579,-35.346,179.369,5.274,149.105
C08725=1231.439,-120.330,-35.356,179.371,5.273,149.105
C08726=1231.434,-120.080,-35.366,179.374,5.274,149.104
C08727=1231.428,-119.829,-35.376,179.376,5.273,149.103
C08728=1231.423,-119.580,-35.386,179.377,5.273,149.103
C08729=1231.418,-119.330,-35.396,179.380,5.274,149.102
C08730=1231.414,-119.080,-35.406,179.382,5.273,149.101
C08731=1231.408,-118.830,-35.415,179.385,5.274,149.101
C08732=1231.402,-118.581,-35.425,179.387,5.273,149.100
C08733=1231.397,-118.331,-35.435,179.390,5.274,149.099
C08734=1231.392,-118.081,-35.446,179.392,5.274,149.098
C08735=1231.387,-117.832,-35.456,179.394,5.274,149.098
C08736=1231.382,-117.582,-35.465,179.396,5.274,149.097
C08737=1231.376,-117.332,-35.475,179.398,5.274,149.096
C08738=1231.371,-117.082,-35.485,179.401,5.274,149.096
C08739=1231.365,-116.832,-35.496,179.403,5.274,149.095
C08740=1231.360,-116.583,-35.505,179.406,5.274,149.094
C08741=1231.355,-116.333,-35.516,179.408,5.274,149.094
C08742=1231.350,-116.083,-35.526,179.410,5.274,149.093
C08743=1231.345,-115.834,-35.536,179.412,5.274,149.092
C08744=1231.340,-115.584,-35.546,179.415,5.274,149.091
C08745=1231.334,-115.334,-35.557,179.417,5.274,149.091
C08746=1231.328,-115.084,-35.566,179.419,5.275,149.090
C08747=1231.324,-114.834,-35.576,179.421,5.274,149.090
C08748=1231.319,-114.585,-35.586,179.424,5.274,149.089
C08749=1231.313,-114.335,-35.596,179.426,5.274,149.088
C08750=1231.308,-114.085,-35.607,179.428,5.274,149.087
C08751=1231.303,-113.836,-35.617,179.431,5.274,149.087
C08752=1231.298,-113.586,-35.627,179.433,5.274,149.086
C08753=1231.293,-113.336,-35.637,179.436,5.274,149.085
C08754=1231.287,-113.086,-35.648,179.438,5.274,149.085
C08755=1231.282,-112.837,-35.657,179.441,5.274,149.084
C08756=1231.277,-112.587,-35.668,179.443,5.274,149.083
C08757=1231.271,-112.337,-35.678,179.445,5.275,149.083
C08758=1231.266,-112.088,-35.688,179.447,5.275,149.082
C08759=1231.261,-111.838,-35.699,179.449,5.274,149.081
C08760=1231.256,-111.588,-35.708,179.452,5.275,149.080
C08761=1231.250,-111.339,-35.719,179.454,5.274,149.080
C08762=1231.245,-111.089,-35.729,179.456,5.275,149.079
C08763=1231.240,-110.839,-35.739,179.459,5.274,149.078
C08764=1231.234,-110.590,-35.750,179.461,5.275,149.078
C08765=1231.230,-110.340,-35.760,179.463,5.274,149.077
C08766=1231.224,-110.090,-35.770,179.466,5.275,149.076
C08767=1231.219,-109.840,-35.780,179.468,5.274,149.075
C08768=1231.214,-109.590,-35.791,179.470,5.275,149.075
C08769=1231.208,-109.341,-35.801,179.472,5.275,149.074
C08770=1231.203,-109.090,-35.811,179.475,5.275,149.074
C08771=1231.198,-108.841,-35.821,179.477,5.275,149.073
C08772=1231.193,-108.591,-35.832,179.479,5.275,149.072
C08773=1231.188,-108.341,-35.842,179.482,5.275,149.071
C08774=1231.182,-108.093,-35.853,179.484,5.275,149.071
C08775=1231.177,-107.842,-35.863,179.487,5.275,149.070
C08776=1231.172,-107.593,-35.873,179.489,5.275,149.069
C08777=1231.167,-107.343,-35.884,179.491,5.275,149.069
C08778=1231.161,-107.093,-35.894,179.494,5.275,149.068
C08779=1231.157,-106.843,-35.904,179.496,5.275,149.067
C08780=1231.151,-106.593,-35.914,179.498,5.275,149.066
C08781=1231.146,-106.344,-35.925,179.500,5.276,149.066
C08782=1231.141,-106.094,-35.936,179.503,5.275,149.065
C08783=1231.136,-105.845,-35.946,179.505,5.276,149.064
C08784=1231.131,-105.595,-35.957,179.507,5.275,149.064
C08785=1231.125,-105.345,-35.967,179.509,5.275,149.063
C08786=1231.120,-105.095,-35.977,179.512,5.276,149.062
C08787=1231.114,-104.845,-35.988,179.514,5.275,149.062
C08788=1231.110,-104.596,-35.999,179.517,5.276,149.061
C08789=1231.104,-104.346,-36.009,179.519,5.275,149.060
C08790=1231.098,-104.097,-36.019,179.522,5.276,149.059
C08791=1231.093,-103.846,-36.030,179.524,5.275,149.059
C08792=1231.089,-103.597,-36.040,179.526,5.276,149.058
C08793=1231.084,-103.347,-36.051,179.529,5.275,149.057
C08794=1231.078,-103.098,-36.061,179.531,5.276,149.057
C08795=1231.073,-102.848,-36.072,179.533,5.275,149.056
C08796=1231.068,-102.598,-36.082,179.535,5.276,149.055
C08797=1231.063,-102.348,-36.093,179.538,5.276,149.055
C08798=1231.057,-102.099,-36.103,179.540,5.276,149.054
C08799=1231.052,-101.849,-36.114,179.542,5.276,149.053
C08800=1231.047,-101.599,-36.124,179.544,5.276,149.053
C08801=1231.042,-101.349,-36.135,179.547,5.276,149.052
C08802=1231.037,-101.100,-36.146,179.549,5.276,149.051
C08803=1231.031,-100.828,-36.157,179.552,5.276,149.050
C08804=1231.026,-100.558,-36.169,179.555,5.276,149.049
C08805=1231.019,-100.287,-36.180,179.557,5.276,149.049
C08806=1231.014,-100.016,-36.192,179.560,5.276,149.048
C08807=1231.009,-99.766,-36.203,179.562,5.276,149.047
C08808=1231.003,-99.517,-36.214,179.565,5.276,149.047
C08809=1230.998,-99.266,-36.224,179.567,5.276,149.046
C08810=1230.993,-99.017,-36.235,179.569,5.276,149.045
C08811=1230.988,-98.767,-36.246,179.571,5.276,149.044
C08812=1230.982,-98.518,-36.256,179.574,5.277,149.044
C08813=1230.977,-98.267,-36.267,179.576,5.276,149.043
C08814=1230.972,-98.018,-36.278,179.579,5.277,149.042
C08815=1230.967,-97.768,-36.288,179.580,5.277,149.042
C08816=1230.962,-97.519,-36.298,179.583,5.277,149.041
C08817=1230.957,-97.269,-36.310,179.585,5.277,149.040
C08818=1230.951,-97.020,-36.320,179.588,5.277,149.040
C08819=1230.947,-96.770,-36.331,179.590,5.277,149.039
C08820=1230.942,-96.520,-36.342,179.592,5.276,149.038
C08821=1230.935,-96.270,-36.352,179.595,5.277,149.038
C08822=1230.930,-96.020,-36.364,179.597,5.277,149.037
C08823=1230.925,-95.771,-36.374,179.600,5.277,149.036
C08824=1230.920,-95.521,-36.385,179.602,5.277,149.035
C08825=1230.915,-95.271,-36.395,179.604,5.277,149.035
C08826=1230.910,-95.022,-36.407,179.606,5.277,149.034
C08827=1230.905,-94.772,-36.417,179.609,5.277,149.033
C08828=1230.900,-94.523,-36.428,179.611,5.277,149.033
C08829=1230.894,-94.272,-36.439,179.614,5.277,149.032
C08830=1230.888,-94.023,-36.450,179.616,5.277,149.031
C08831=1230.884,-93.773,-36.461,179.619,5.277,149.030
C08832=1230.879,-93.523,-36.471,179.621,5.277,149.030
C08833=1230.873,-93.274,-36.482,179.623,5.277,149.029
C08834=1230.868,-93.024,-36.493,179.625,5.277,149.028
C08835=1230.863,-92.775,-36.504,179.628,5.278,149.028
C08836=1230.857,-92.524,-36.515,179.630,5.277,149.027
C08837=1230.853,-92.274,-36.526,179.633,5.278,149.026
C08838=1230.847,-92.026,-36.537,179.635,5.277,149.025
C08839=1230.842,-91.775,-36.548,179.638,5.278,149.025
C08840=1230.837,-91.526,-36.559,179.639,5.278,149.024
C08841=1230.831,-91.276,-36.570,179.642,5.278,149.024
C08842=1230.827,-91.026,-36.581,179.644,5.278,149.023
C08843=1230.821,-90.777,-36.591,179.647,5.278,149.022
C08844=1230.816,-90.527,-36.603,179.649,5.278,149.021
C08845=1230.811,-90.277,-36.613,179.652,5.278,149.021
C08846=1230.805,-90.028,-36.625,179.654,5.278,149.020
C08847=1230.801,-89.778,-36.636,179.656,5.278,149.019
C08848=1230.796,-89.528,-36.647,179.658,5.278,149.019
C08849=1230.790,-89.279,-36.658,179.661,5.279,149.018
C08850=1230.785,-89.028,-36.669,179.663,5.278,149.017
C08851=1230.780,-88.779,-36.680,179.665,5.278,149.016
C08852=1230.775,-88.530,-36.691,179.668,5.278,149.016
C08853=1230.770,-88.279,-36.702,179.670,5.278,149.015
C08854=1230.764,-88.029,-36.713,179.673,5.278,149.014
C08855=1230.759,-87.781,-36.724,179.675,5.278,149.014
C08856=1230.754,-87.530,-36.735,179.677,5.279,149.013
C08857=1230.749,-87.281,-36.746,179.680,5.278,149.012
C08858=1230.743,-87.031,-36.758,179.682,5.279,149.011
C08859=1230.738,-86.781,-36.768,179.684,5.278,149.011
C08860=1230.733,-86.532,-36.780,179.687,5.279,149.010
C08861=1230.727,-86.282,-36.791,179.689,5.278,149.009
C08862=1230.722,-86.032,-36.802,179.692,5.279,149.009
C08863=1230.718,-85.782,-36.813,179.694,5.278,149.008
C08864=1230.713,-85.533,-36.824,179.696,5.279,149.007
C08865=1230.707,-85.283,-36.835,179.699,5.279,149.007
C08866=1230.702,-85.033,-36.846,179.701,5.279,149.006
C08867=1230.697,-84.784,-36.858,179.703,5.279,149.005
C08868=1230.691,-84.534,-36.869,179.706,5.279,149.004
C08869=1230.686,-84.284,-36.880,179.708,5.279,149.004
C08870=1230.682,-84.035,-36.891,179.711,5.279,149.003
C08871=1230.676,-83.785,-36.903,179.713,5.279,149.002
C08872=1230.671,-83.536,-36.914,179.716,5.279,149.002
C08873=1230.666,-83.285,-36.924,179.718,5.279,149.001
C08874=1230.660,-83.036,-36.936,179.720,5.279,149.000
C08875=1230.656,-82.786,-36.948,179.722,5.279,148.999
C08876=1230.650,-82.537,-36.959,179.725,5.280,148.999
C08877=1230.645,-82.287,-36.970,179.727,5.279,148.998
C08878=1230.640,-82.037,-36.981,179.730,5.280,148.997
C08879=1230.635,-81.787,-36.993,179.732,5.279,148.997
C08880=1230.629,-81.538,-37.004,179.735,5.280,148.996
C08881=1230.625,-81.288,-37.015,179.737,5.279,148.995
C08882=1230.619,-81.038,-37.027,179.739,5.280,148.994
C08883=1230.614,-80.789,-37.038,179.741,5.280,148.994
C08884=1230.608,-80.539,-37.049,179.744,5.280,148.993
C08885=1230.603,-80.289,-37.060,179.746,5.280,148.992
C08886=1230.599,-80.040,-37.072,179.749,5.280,148.992
C08887=1230.593,-79.790,-37.084,179.751,5.280,148.991
C08888=1230.589,-79.540,-37.095,179.754,5.280,148.990
C08889=1230.583,-79.291,-37.106,179.756,5.280,148.989
C08890=1230.578,-79.041,-37.118,179.758,5.280,148.989
C08891=1230.572,-78.791,-37.130,179.760,5.280,148.988
C08892=1230.568,-78.542,-37.141,179.763,5.280,148.987
C08893=1230.562,-78.291,-37.152,179.766,5.281,148.987
C08894=1230.557,-78.042,-37.163,179.768,5.281,148.986
C08895=1230.552,-77.793,-37.174,179.771,5.281,148.985
C08896=1230.547,-77.543,-37.186,179.773,5.281,148.985
C08897=1230.542,-77.293,-37.197,179.775,5.281,148.984
C08898=1230.537,-77.043,-37.209,179.777,5.281,148.983
C08899=1230.532,-76.793,-37.221,179.780,5.281,148.982
C08900=1230.526,-76.544,-37.232,179.782,5.281,148.982
C08901=1230.521,-76.295,-37.243,179.785,5.281,148.981
C08902=1230.516,-76.045,-37.255,179.787,5.281,148.980
C08903=1230.511,-75.795,-37.267,179.790,5.281,148.980
C08904=1230.506,-75.545,-37.278,179.792,5.281,148.979
C08905=1230.500,-75.296,-37.289,179.794,5.282,148.978
C08906=1230.495,-75.046,-37.301,179.796,5.281,148.977
C08907=1230.489,-74.775,-37.314,179.799,5.282,148.977
C08908=1230.484,-74.505,-37.326,179.801,5.281,148.976
C08909=1230.478,-74.235,-37.339,179.804,5.282,148.975
C08910=1230.472,-73.964,-37.351,179.807,5.282,148.974
C08911=1230.468,-73.715,-37.363,179.809,5.282,148.974
C08912=1230.462,-73.465,-37.375,179.812,5.282,148.973
C08913=1230.457,-73.216,-37.385,179.814,5.282,148.972
C08914=1230.452,-72.966,-37.398,179.817,5.282,148.972
C08915=1230.446,-72.717,-37.410,179.819,5.282,148.971
C08916=1230.442,-72.467,-37.421,179.821,5.282,148.970
C08917=1230.436,-72.217,-37.433,179.823,5.282,148.969
C08918=1230.432,-71.967,-37.444,179.826,5.282,148.969
C08919=1230.426,-71.717,-37.456,179.828,5.282,148.968
C08920=1230.421,-71.467,-37.468,179.831,5.283,148.967
C08921=1230.415,-71.219,-37.479,179.833,5.282,148.967
C08922=1230.410,-70.969,-37.491,179.836,5.283,148.966
C08923=1230.405,-70.719,-37.502,179.838,5.283,148.965
C08924=1230.400,-70.470,-37.515,179.840,5.283,148.964
C08925=1230.395,-70.220,-37.527,179.843,5.283,148.964
C08926=1230.390,-69.970,-37.538,179.845,5.283,148.963
C08927=1230.385,-69.720,-37.550,179.848,5.283,148.962
C08928=1230.379,-69.470,-37.562,179.850,5.283,148.962
C08929=1230.375,-69.221,-37.573,179.853,5.284,148.961
C08930=1230.369,-68.971,-37.585,179.855,5.283,148.960
C08931=1230.365,-68.722,-37.597,179.857,5.284,148.959
C08932=1230.359,-68.472,-37.609,179.859,5.283,148.959
C08933=1230.353,-68.222,-37.620,179.862,5.284,148.958
C08934=1230.349,-67.973,-37.632,179.864,5.283,148.957
C08935=1230.343,-67.723,-37.644,179.867,5.284,148.957
C08936=1230.338,-67.474,-37.656,179.869,5.284,148.956
C08937=1230.333,-67.224,-37.667,179.872,5.284,148.955
C08938=1230.328,-66.974,-37.679,179.874,5.284,148.955
C08939=1230.322,-66.724,-37.691,179.876,5.284,148.954
C08940=1230.317,-66.475,-37.704,179.879,5.285,148.953
C08941=1230.313,-66.225,-37.715,179.881,5.284,148.952
C08942=1230.307,-65.975,-37.727,179.884,5.285,148.952
C08943=1230.302,-65.725,-37.739,179.886,5.284,148.951
C08944=1230.297,-65.476,-37.751,179.889,5.285,148.950
C08945=1230.292,-65.226,-37.763,179.891,5.285,148.950
C08946=1230.287,-64.976,-37.775,179.893,5.285,148.949
C08947=1230.281,-64.726,-37.787,179.895,5.285,148.948
C08948=1230.277,-64.477,-37.799,179.898,5.285,148.947
C08949=1230.271,-64.228,-37.810,179.900,5.285,148.947
C08950=1230.266,-63.978,-37.822,179.903,5.285,148.946
C08951=1230.261,-63.728,-37.835,179.905,5.285,148.945
C08952=1230.256,-63.479,-37.846,179.908,5.285,148.945
C08953=1230.251,-63.229,-37.858,179.910,5.286,148.944
C08954=1230.246,-62.979,-37.871,179.912,5.286,148.943
C08955=1230.240,-62.729,-37.883,179.915,5.286,148.943
C08956=1230.235,-62.480,-37.894,179.917,5.286,148.942
C08957=1230.230,-62.231,-37.906,179.920,5.286,148.941
C08958=1230.225,-61.981,-37.918,179.922,5.286,148.940
C08959=1230.220,-61.731,-37.931,179.925,5.286,148.940
C08960=1230.214,-61.481,-37.943,179.927,5.286,148.939
C08961=1230.210,-61.232,-37.954,179.929,5.286,148.938
C08962=1230.204,-60.982,-37.967,179.931,5.286,148.938
C08963=1230.199,-60.732,-37.979,179.934,5.287,148.937
C08964=1230.194,-60.483,-37.991,179.937,5.287,148.936
C08965=1230.188,-60.233,-38.003,179.939,5.287,148.935
C08966=1230.184,-59.984,-38.014,179.941,5.287,148.935
C08967=1230.179,-59.734,-38.027,179.944,5.287,148.934
C08968=1230.174,-59.484,-38.039,179.946,5.287,148.933
C08969=1230.169,-59.234,-38.052,179.948,5.287,148.933
C08970=1230.163,-58.984,-38.064,179.951,5.288,148.932
C08971=1230.158,-58.735,-38.076,179.953,5.287,148.931
C08972=1230.153,-58.485,-38.088,179.956,5.288,148.931
C08973=1230.148,-58.236,-38.100,179.958,5.287,148.930
C08974=1230.143,-57.986,-38.112,179.961,5.287,148.929
C08975=1230.138,-57.737,-38.125,179.964,5.288,148.928
C08976=1230.132,-57.487,-38.137,179.966,5.288,148.927
C08977=1230.127,-57.238,-38.149,179.968,5.288,148.927
C08978=1230.122,-56.988,-38.161,179.970,5.288,148.926
C08979=1230.117,-56.738,-38.174,179.973,5.288,148.925
C08980=1230.113,-56.488,-38.185,179.975,5.288,148.925
C08981=1230.107,-56.239,-38.198,179.978,5.288,148.924
C08982=1230.102,-55.989,-38.210,179.980,5.288,148.923
C08983=1230.097,-55.739,-38.222,179.983,5.288,148.923
C08984=1230.091,-55.489,-38.234,179.985,5.289,148.922
C08985=1230.086,-55.240,-38.247,179.987,5.289,148.921
C08986=1230.081,-54.990,-38.259,179.990,5.289,148.920
C08987=1230.076,-54.741,-38.271,179.992,5.289,148.920
C08988=1230.071,-54.492,-38.284,179.995,5.289,148.919
C08989=1230.066,-54.241,-38.296,179.997,5.289,148.918
C08990=1230.061,-53.992,-38.309,180.000,5.289,148.918
C08991=1230.055,-53.742,-38.321,-179.998,5.290,148.917
C08992=1230.051,-53.493,-38.333,-179.996,5.290,148.916
C08993=1230.046,-53.243,-38.345,-179.993,5.290,148.916
C08994=1230.040,-52.993,-38.357,-179.991,5.290,148.915
C08995=1230.035,-52.744,-38.370,-179.988,5.290,148.914
C08996=1230.031,-52.494,-38.383,-179.986,5.290,148.913
C08997=1230.025,-52.244,-38.395,-179.983,5.290,148.913
C08998=1230.020,-51.995,-38.407,-179.981,5.290,148.912
C08999=1230.015,-51.746,-38.420,-179.979,5.291,148.911
C09000=1230.010,-51.496,-38.432,-179.976,5.291,148.911
C09001=1230.004,-51.246,-38.444,-179.974,5.291,148.910
C09002=1230.000,-50.996,-38.457,-179.971,5.291,148.909
C09003=1229.995,-50.746,-38.469,-179.969,5.291,148.908
C09004=1229.989,-50.497,-38.482,-179.967,5.291,148.908
C09005=1229.984,-50.248,-38.494,-179.964,5.291,148.907
C09006=1229.979,-49.998,-38.506,-179.962,5.291,148.906
C09007=1229.974,-49.748,-38.519,-179.959,5.292,148.906
C09008=1229.969,-49.498,-38.532,-179.957,5.292,148.905
C09009=1229.963,-49.249,-38.545,-179.954,5.292,148.904
C09010=1229.958,-48.999,-38.557,-179.952,5.291,148.903
C09011=1229.953,-48.729,-38.571,-179.949,5.292,148.903
C09012=1229.947,-48.460,-38.584,-179.946,5.292,148.902
C09013=1229.942,-48.190,-38.598,-179.944,5.292,148.901
C09014=1229.936,-47.920,-38.611,-179.941,5.292,148.900
C09015=1229.931,-47.670,-38.624,-179.939,5.293,148.900
C09016=1229.926,-47.421,-38.636,-179.936,5.292,148.899
C09017=1229.921,-47.172,-38.649,-179.934,5.293,148.898
C09018=1229.916,-46.921,-38.661,-179.932,5.292,148.897
C09019=1229.911,-46.672,-38.674,-179.929,5.293,148.897
C09020=1229.906,-46.422,-38.686,-179.926,5.293,148.896
C09021=1229.900,-46.173,-38.700,-179.924,5.293,148.895
C09022=1229.895,-45.923,-38.713,-179.922,5.294,148.895
C09023=1229.890,-45.674,-38.725,-179.920,5.293,148.894
C09024=1229.885,-45.424,-38.737,-179.917,5.294,148.893
C09025=1229.880,-45.174,-38.750,-179.914,5.294,148.893
C09026=1229.875,-44.924,-38.763,-179.912,5.294,148.892
C09027=1229.870,-44.675,-38.775,-179.909,5.294,148.891
C09028=1229.864,-44.425,-38.788,-179.907,5.294,148.890
C09029=1229.859,-44.176,-38.801,-179.905,5.295,148.890
C09030=1229.855,-43.926,-38.814,-179.903,5.294,148.889
C09031=1229.849,-43.677,-38.827,-179.900,5.295,148.888
C09032=1229.844,-43.427,-38.839,-179.897,5.295,148.888
C09033=1229.840,-43.177,-38.851,-179.895,5.295,148.887
C09034=1229.834,-42.927,-38.865,-179.893,5.295,148.886
C09035=1229.829,-42.678,-38.877,-179.890,5.295,148.886
C09036=1229.823,-42.428,-38.890,-179.888,5.296,148.885
C09037=1229.819,-42.178,-38.903,-179.885,5.296,148.884
C09038=1229.814,-41.929,-38.915,-179.883,5.296,148.883
C09039=1229.808,-41.679,-38.929,-179.880,5.296,148.883
C09040=1229.803,-41.429,-38.942,-179.878,5.296,148.882
C09041=1229.798,-41.180,-38.954,-179.875,5.296,148.881
C09042=1229.793,-40.931,-38.967,-179.872,5.297,148.880
C09043=1229.789,-40.681,-38.980,-179.870,5.296,148.880
C09044=1229.783,-40.431,-38.993,-179.868,5.297,148.879
C09045=1229.778,-40.182,-39.006,-179.866,5.296,148.878
C09046=1229.773,-39.933,-39.018,-179.863,5.297,148.878
C09047=1229.768,-39.683,-39.031,-179.860,5.297,148.877
C09048=1229.762,-39.433,-39.044,-179.858,5.297,148.876
C09049=1229.757,-39.184,-39.057,-179.856,5.298,148.876
C09050=1229.752,-38.934,-39.070,-179.853,5.297,148.875
C09051=1229.747,-38.684,-39.083,-179.851,5.298,148.874
C09052=1229.742,-38.434,-39.096,-179.848,5.298,148.873
C09053=1229.737,-38.185,-39.109,-179.846,5.298,148.873
C09054=1229.732,-37.935,-39.121,-179.843,5.298,148.872
C09055=1229.727,-37.685,-39.134,-179.841,5.298,148.871
C09056=1229.721,-37.436,-39.147,-179.839,5.299,148.871
C09057=1229.716,-37.186,-39.160,-179.836,5.299,148.870
C09058=1229.712,-36.937,-39.174,-179.834,5.299,148.869
C09059=1229.706,-36.687,-39.187,-179.831,5.299,148.869
C09060=1229.701,-36.438,-39.200,-179.829,5.299,148.868
C09061=1229.697,-36.188,-39.212,-179.827,5.299,148.867
C09062=1229.691,-35.938,-39.226,-179.824,5.300,148.866
C09063=1229.686,-35.688,-39.239,-179.822,5.300,148.866
C09064=1229.681,-35.439,-39.251,-179.819,5.300,148.865
C09065=1229.675,-35.189,-39.264,-179.816,5.301,148.864
C09066=1229.671,-34.940,-39.278,-179.814,5.300,148.864
C09067=1229.666,-34.691,-39.291,-179.812,5.301,148.863
C09068=1229.660,-34.441,-39.304,-179.810,5.300,148.862
C09069=1229.656,-34.191,-39.317,-179.807,5.301,148.862
C09070=1229.650,-33.941,-39.330,-179.804,5.301,148.861
C09071=1229.645,-33.691,-39.343,-179.802,5.301,148.860
C09072=1229.640,-33.443,-39.356,-179.799,5.301,148.859
C09073=1229.635,-33.192,-39.370,-179.797,5.301,148.858
C09074=1229.630,-32.943,-39.383,-179.794,5.301,148.858
C09075=1229.625,-32.694,-39.395,-179.792,5.302,148.857
C09076=1229.620,-32.443,-39.409,-179.790,5.302,148.856
C09077=1229.615,-32.195,-39.422,-179.787,5.302,148.856
C09078=1229.609,-31.944,-39.436,-179.784,5.303,148.855
C09079=1229.604,-31.695,-39.448,-179.782,5.302,148.854
C09080=1229.599,-31.445,-39.462,-179.779,5.303,148.854
C09081=1229.594,-31.196,-39.475,-179.777,5.303,148.853
C09082=1229.589,-30.947,-39.488,-179.775,5.303,148.852
C09083=1229.584,-30.696,-39.501,-179.772,5.304,148.852
C09084=1229.579,-30.448,-39.515,-179.770,5.303,148.851
C09085=1229.574,-30.197,-39.528,-179.767,5.304,148.850
C09086=1229.569,-29.948,-39.541,-179.765,5.304,148.849
C09087=1229.563,-29.698,-39.554,-179.763,5.304,148.849
C09088=1229.559,-29.449,-39.568,-179.760,5.304,148.848
C09089=1229.553,-29.199,-39.581,-179.758,5.304,148.847
C09090=1229.548,-28.949,-39.594,-179.755,5.305,148.847
C09091=1229.544,-28.700,-39.607,-179.753,5.305,148.846
C09092=1229.538,-28.450,-39.621,-179.750,5.305,148.845
C09093=1229.534,-28.200,-39.634,-179.748,5.305,148.845
C09094=1229.528,-27.951,-39.647,-179.745,5.306,148.844
C09095=1229.524,-27.701,-39.660,-179.743,5.306,148.843
C09096=1229.518,-27.452,-39.674,-179.740,5.306,148.842
C09097=1229.513,-27.202,-39.687,-179.738,5.306,148.842
C09098=1229.508,-26.953,-39.701,-179.736,5.306,148.841
C09099=1229.503,-26.703,-39.714,-179.733,5.307,148.840
C09100=1229.498,-26.454,-39.727,-179.731,5.306,148.840
C09101=1229.493,-26.204,-39.742,-179.728,5.307,148.839
C09102=1229.487,-25.955,-39.754,-179.726,5.307,148.838
C09103=1229.482,-25.704,-39.768,-179.723,5.307,148.837
C09104=1229.477,-25.455,-39.781,-179.720,5.307,148.837
C09105=1229.472,-25.205,-39.795,-179.718,5.308,148.836
C09106=1229.467,-24.956,-39.808,-179.716,5.307,148.835
C09107=1229.462,-24.706,-39.822,-179.713,5.308,148.835
C09108=1229.457,-24.457,-39.835,-179.710,5.308,148.834
C09109=1229.452,-24.207,-39.848,-179.708,5.308,148.833
C09110=1229.447,-23.958,-39.862,-179.706,5.309,148.832
C09111=1229.442,-23.708,-39.875,-179.703,5.308,148.832
C09112=1229.437,-23.458,-39.890,-179.701,5.309,148.831
C09113=1229.432,-23.209,-39.902,-179.698,5.309,148.830
C09114=1229.427,-22.959,-39.917,-179.696,5.309,148.830
C09115=1229.420,-22.690,-39.930,-179.693,5.310,148.829
C09116=1229.416,-22.421,-39.945,-179.691,5.310,148.828
C09117=1229.410,-22.151,-39.960,-179.688,5.310,148.827
C09118=1229.405,-21.882,-39.975,-179.685,5.311,148.827
C09119=1229.399,-21.632,-39.988,-179.683,5.310,148.826
C09120=1229.395,-21.383,-40.002,-179.680,5.311,148.825
C09121=1229.389,-21.134,-40.016,-179.678,5.311,148.825
C09122=1229.385,-20.884,-40.029,-179.675,5.311,148.824
C09123=1229.380,-20.634,-40.043,-179.673,5.312,148.823
C09124=1229.374,-20.385,-40.056,-179.671,5.311,148.822
C09125=1229.370,-20.135,-40.070,-179.668,5.312,148.822
C09126=1229.364,-19.886,-40.083,-179.665,5.312,148.821
C09127=1229.359,-19.636,-40.097,-179.663,5.312,148.820
C09128=1229.355,-19.387,-40.111,-179.661,5.313,148.820
C09129=1229.349,-19.137,-40.124,-179.658,5.313,148.819
C09130=1229.344,-18.887,-40.138,-179.656,5.313,148.818
C09131=1229.339,-18.637,-40.153,-179.653,5.313,148.818
